Yaskawa INFORM job: u_tourne3TRJ1.JBI

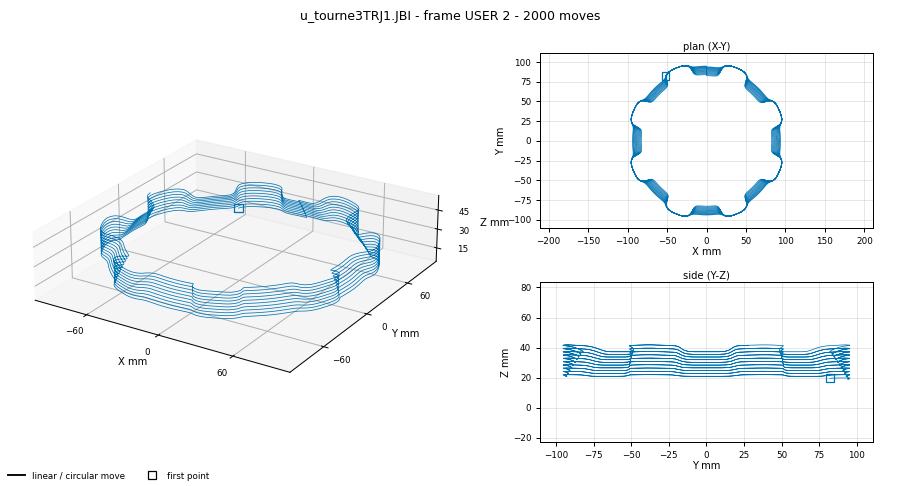
[picture p0: tool path of u_tourne3TRJ1.JBI in frame USER 2, 2000 of 2000 moves have a stored position in this frame; points joined in program order, loops and branches not executed]
/JOB
//NAME u_tourne3TRJ1
///FOLDERNAME DEMO
//POS
///NPOS 2000,0,2000,0,0,0
///USER 2
///TOOL 7
///POSTYPE USER
///RECTAN
///RCONF 1,0,0,0,0,0,0,0,0,0,0,0,0,0,0,0,0,0,0,0,0,0,0,0
C00000=-51.961,81.931,19.493,173.8545,9.2440,-3657.6170
C00001=-51.163,83.502,19.627,176.6033,6.2165,-3658.5035
C00002=-49.917,85.194,19.692,178.7206,4.0258,-3659.6330
C00003=-47.874,87.106,19.726,179.6780,1.7463,-3661.2065
C00004=-45.272,88.975,19.753,179.9712,0.2718,-3663.0322
C00005=-42.449,90.515,19.780,179.9981,0.0768,-3664.8747
C00006=-39.659,91.796,19.798,179.9970,0.0075,-3666.6340
C00007=-36.867,92.953,19.798,179.9968,0.0074,-3668.3657
C00008=-33.988,94.020,19.780,-179.9962,0.0778,-3670.1252
C00009=-30.903,94.927,19.753,-179.9766,0.2756,-3671.9676
C00010=-27.741,95.446,19.726,-179.6779,1.7445,-3673.7937
C00011=-24.945,95.538,19.692,-178.7208,4.0294,-3675.3667
C00012=-22.867,95.222,19.627,-176.6046,6.2189,-3676.4965
C00013=-21.192,94.676,19.493,-173.8561,9.2462,-3677.3831
C00014=-19.540,94.146,19.309,-171.9611,14.9094,-3678.2747
C00015=-17.528,93.824,19.120,-173.2655,21.6484,-3679.4181
C00016=-14.592,93.857,18.976,-177.3137,25.8724,-3681.1629
C00017=-10.190,94.262,18.917,-179.5911,27.0185,-3683.8301
C00018=-5.317,94.652,18.914,179.9702,27.0874,-3686.7848
C00019=0.000,94.804,18.916,-180.0000,27.0775,-3690.0000
C00020=0.000,93.772,20.859,-180.0000,28.8281,-3690.0000
C00021=5.223,93.624,20.857,-179.9587,28.8401,-3693.1930
C00022=10.031,93.243,20.860,179.4696,28.7637,-3696.1402
C00023=14.399,92.874,20.935,176.5083,27.4530,-3698.8129
C00024=17.292,92.935,21.118,171.4736,22.1760,-3700.5402
C00025=19.271,93.399,21.361,170.6019,14.0567,-3701.6582
C00026=20.902,94.108,21.598,173.3176,8.0331,-3702.5225
C00027=22.556,94.852,21.773,176.3408,5.3244,-3703.3766
C00028=24.607,95.353,21.858,178.5800,3.6143,-3704.4702
C00029=27.423,95.407,21.902,179.6582,1.5415,-3706.0363
C00030=30.651,94.973,21.938,179.9852,0.1578,-3707.8866
C00031=33.828,94.073,21.973,-179.9998,0.0671,-3709.7782
C00032=36.813,92.974,21.997,179.9979,0.0053,-3711.6011
C00033=39.712,91.773,21.997,-179.9970,0.0075,-3713.3991
C00034=42.599,90.440,21.973,179.9991,0.0692,-3715.2213
C00035=45.483,88.829,21.938,-179.9836,0.1565,-3717.1138
C00036=48.072,86.854,21.902,-179.6591,1.5379,-3718.9637
C00037=50.025,84.825,21.858,-178.5802,3.6128,-3720.5297
C00038=51.121,83.020,21.773,-176.3413,5.3283,-3721.6234
C00039=51.765,81.324,21.598,-173.3148,8.0333,-3722.4779
C00040=52.416,79.670,21.361,-170.5989,14.0579,-3723.3415
C00041=53.488,77.942,21.118,-171.4764,22.1779,-3724.4600
C00042=55.491,75.854,20.935,-176.5044,27.4539,-3726.1873
C00043=58.840,73.026,20.860,-179.4708,28.7627,-3728.8598
C00044=62.509,69.895,20.857,179.9582,28.8407,-3731.8071
C00045=66.307,66.307,20.859,180.0000,28.8305,-3735.0000
C00046=69.895,62.509,20.857,-179.9582,28.8407,-3738.1929
C00047=73.026,58.840,20.860,179.4708,28.7627,-3741.1402
C00048=75.854,55.491,20.935,176.5044,27.4539,-3743.8127
C00049=77.942,53.488,21.118,171.4764,22.1779,-3745.5400
C00050=79.670,52.416,21.361,170.5989,14.0579,-3746.6585
C00051=81.324,51.765,21.598,173.3148,8.0333,-3747.5221
C00052=83.020,51.121,21.773,176.3413,5.3283,-3748.3766
C00053=84.825,50.025,21.858,178.5802,3.6128,-3749.4703
C00054=86.854,48.072,21.902,179.6591,1.5379,-3751.0363
C00055=88.829,45.483,21.938,179.9836,0.1565,-3752.8862
C00056=90.440,42.599,21.973,-179.9991,0.0692,-3754.7787
C00057=91.773,39.712,21.997,179.9970,0.0075,-3756.6009
C00058=92.974,36.813,21.997,-179.9979,0.0053,-3758.3989
C00059=94.073,33.828,21.973,179.9998,0.0671,-3760.2218
C00060=94.973,30.651,21.938,-179.9852,0.1578,-3762.1134
C00061=95.407,27.423,21.902,-179.6582,1.5415,-3763.9637
C00062=95.353,24.607,21.858,-178.5800,3.6143,-3765.5298
C00063=94.852,22.556,21.773,-176.3408,5.3244,-3766.6234
C00064=94.108,20.902,21.598,-173.3176,8.0331,-3767.4775
C00065=93.399,19.271,21.361,-170.6019,14.0567,-3768.3418
C00066=92.935,17.292,21.118,-171.4736,22.1760,-3769.4598
C00067=92.874,14.399,20.935,-176.5083,27.4530,-3771.1871
C00068=93.243,10.031,20.860,-179.4696,28.7637,-3773.8598
C00069=93.624,5.223,20.857,179.9587,28.8401,-3776.8070
C00070=93.772,0.000,20.859,180.0000,28.8281,-3780.0000
C00071=93.624,-5.223,20.857,-179.9587,28.8401,-3783.1930
C00072=93.243,-10.031,20.860,179.4696,28.7637,-3786.1402
C00073=92.875,-14.399,20.935,176.5083,27.4530,-3788.8128
C00074=92.935,-17.292,21.118,171.4736,22.1760,-3790.5402
C00075=93.399,-19.271,21.361,170.6019,14.0567,-3791.6582
C00076=94.108,-20.902,21.598,173.3176,8.0331,-3792.5225
C00077=94.852,-22.556,21.773,176.3408,5.3244,-3793.3766
C00078=95.353,-24.607,21.858,178.5800,3.6143,-3794.4702
C00079=95.407,-27.423,21.902,179.6582,1.5415,-3796.0363
C00080=94.973,-30.651,21.938,179.9852,0.1578,-3797.8866
C00081=94.073,-33.828,21.973,-179.9998,0.0671,-3799.7782
C00082=92.974,-36.813,21.997,179.9979,0.0053,-3801.6011
C00083=91.773,-39.712,21.997,-179.9970,0.0075,-3803.3991
C00084=90.440,-42.599,21.973,179.9991,0.0692,-3805.2213
C00085=88.829,-45.483,21.938,-179.9836,0.1565,-3807.1138
C00086=86.854,-48.072,21.902,-179.6591,1.5379,-3808.9637
C00087=84.825,-50.025,21.858,-178.5802,3.6128,-3810.5297
C00088=83.020,-51.121,21.773,-176.3413,5.3283,-3811.6234
C00089=81.324,-51.765,21.598,-173.3148,8.0333,-3812.4779
C00090=79.670,-52.416,21.361,-170.5989,14.0579,-3813.3415
C00091=77.942,-53.488,21.118,-171.4764,22.1779,-3814.4600
C00092=75.854,-55.491,20.935,-176.5044,27.4539,-3816.1873
C00093=73.026,-58.840,20.860,-179.4708,28.7627,-3818.8598
C00094=69.895,-62.509,20.857,179.9582,28.8407,-3821.8071
C00095=66.307,-66.307,20.859,-180.0000,28.8305,-3825.0000
C00096=62.509,-69.895,20.857,-179.9582,28.8407,-3828.1929
C00097=58.840,-73.026,20.860,179.4708,28.7627,-3831.1402
C00098=55.491,-75.854,20.935,176.5044,27.4539,-3833.8127
C00099=53.488,-77.942,21.118,171.4764,22.1779,-3835.5400
C00100=52.416,-79.670,21.361,170.5989,14.0579,-3836.6585
C00101=51.765,-81.324,21.598,173.3148,8.0333,-3837.5221
C00102=51.121,-83.020,21.773,176.3413,5.3283,-3838.3766
C00103=50.025,-84.825,21.858,178.5802,3.6128,-3839.4703
C00104=48.072,-86.854,21.902,179.6591,1.5379,-3841.0363
C00105=45.483,-88.829,21.938,179.9836,0.1565,-3842.8862
C00106=42.599,-90.440,21.973,-179.9991,0.0692,-3844.7787
C00107=39.712,-91.773,21.997,179.9970,0.0075,-3846.6009
C00108=36.813,-92.974,21.997,-179.9979,0.0053,-3848.3989
C00109=33.828,-94.073,21.973,179.9998,0.0671,-3850.2218
C00110=30.651,-94.973,21.938,-179.9852,0.1578,-3852.1134
C00111=27.423,-95.407,21.902,-179.6582,1.5415,-3853.9637
C00112=24.607,-95.353,21.858,-178.5800,3.6143,-3855.5298
C00113=22.556,-94.852,21.773,-176.3408,5.3244,-3856.6234
C00114=20.902,-94.108,21.598,-173.3176,8.0331,-3857.4775
C00115=19.271,-93.399,21.361,-170.6019,14.0567,-3858.3418
C00116=17.292,-92.935,21.118,-171.4736,22.1760,-3859.4598
C00117=14.399,-92.874,20.935,-176.5083,27.4530,-3861.1871
C00118=10.031,-93.243,20.860,-179.4696,28.7637,-3863.8598
C00119=5.223,-93.624,20.857,179.9587,28.8401,-3866.8070
C00120=0.000,-93.772,20.859,-180.0000,28.8281,-3870.0000
C00121=0.000,-93.772,20.859,-180.0000,28.8281,-3870.0000
C00122=-5.223,-93.624,20.857,-179.9587,28.8401,-3873.1930
C00123=-10.031,-93.243,20.860,179.4696,28.7637,-3876.1402
C00124=-14.399,-92.875,20.935,176.5083,27.4530,-3878.8128
C00125=-17.292,-92.935,21.118,171.4736,22.1760,-3880.5402
C00126=-19.271,-93.399,21.361,170.6019,14.0567,-3881.6582
C00127=-20.902,-94.108,21.598,173.3176,8.0331,-3882.5225
C00128=-22.556,-94.852,21.773,176.3408,5.3244,-3883.3766
C00129=-24.607,-95.353,21.858,178.5800,3.6143,-3884.4702
C00130=-27.423,-95.407,21.902,179.6582,1.5415,-3886.0363
C00131=-30.651,-94.973,21.938,179.9852,0.1578,-3887.8866
C00132=-33.828,-94.073,21.973,-179.9998,0.0671,-3889.7782
C00133=-36.813,-92.974,21.997,179.9979,0.0053,-3891.6011
C00134=-39.712,-91.773,21.997,-179.9970,0.0075,-3893.3991
C00135=-42.599,-90.440,21.973,179.9991,0.0692,-3895.2213
C00136=-45.483,-88.829,21.938,-179.9836,0.1565,-3897.1138
C00137=-48.072,-86.854,21.902,-179.6591,1.5379,-3898.9637
C00138=-50.025,-84.825,21.858,-178.5802,3.6128,-3900.5297
C00139=-51.121,-83.020,21.773,-176.3413,5.3283,-3901.6234
C00140=-51.765,-81.324,21.598,-173.3148,8.0333,-3902.4779
C00141=-52.416,-79.670,21.361,-170.5989,14.0579,-3903.3415
C00142=-53.488,-77.942,21.118,-171.4764,22.1779,-3904.4600
C00143=-55.491,-75.854,20.935,-176.5044,27.4539,-3906.1873
C00144=-58.840,-73.026,20.860,-179.4708,28.7627,-3908.8598
C00145=-62.509,-69.895,20.857,179.9582,28.8407,-3911.8071
C00146=-66.307,-66.307,20.859,-180.0000,28.8305,-3915.0000
C00147=-69.895,-62.509,20.857,-179.9582,28.8407,-3918.1929
C00148=-73.026,-58.840,20.860,179.4708,28.7627,-3921.1402
C00149=-75.854,-55.491,20.935,176.5044,27.4539,-3923.8127
C00150=-77.942,-53.488,21.118,171.4764,22.1779,-3925.5400
C00151=-79.670,-52.416,21.361,170.5989,14.0579,-3926.6585
C00152=-81.324,-51.765,21.598,173.3148,8.0333,-3927.5221
C00153=-83.020,-51.121,21.773,176.3413,5.3283,-3928.3766
C00154=-84.825,-50.025,21.858,178.5802,3.6128,-3929.4703
C00155=-86.854,-48.072,21.902,179.6591,1.5379,-3931.0363
C00156=-88.829,-45.483,21.938,179.9836,0.1565,-3932.8862
C00157=-90.440,-42.599,21.973,-179.9991,0.0692,-3934.7787
C00158=-91.773,-39.712,21.997,179.9970,0.0075,-3936.6009
C00159=-92.974,-36.813,21.997,-179.9979,0.0053,-3938.3989
C00160=-94.073,-33.828,21.973,179.9998,0.0671,-3940.2218
C00161=-94.973,-30.651,21.938,-179.9852,0.1578,-3942.1134
C00162=-95.407,-27.423,21.902,-179.6582,1.5415,-3943.9637
C00163=-95.353,-24.607,21.858,-178.5800,3.6143,-3945.5298
C00164=-94.852,-22.556,21.773,-176.3408,5.3244,-3946.6234
C00165=-94.108,-20.902,21.598,-173.3176,8.0331,-3947.4775
C00166=-93.399,-19.271,21.361,-170.6019,14.0567,-3948.3418
C00167=-92.935,-17.292,21.118,-171.4736,22.1760,-3949.4598
C00168=-92.874,-14.399,20.935,-176.5083,27.4530,-3951.1871
C00169=-93.243,-10.031,20.860,-179.4696,28.7637,-3953.8598
C00170=-93.624,-5.223,20.857,179.9587,28.8401,-3956.8070
C00171=-93.772,0.000,20.859,180.0000,28.8281,-3960.0000
C00172=-93.624,5.223,20.857,-179.9587,28.8401,-3963.1930
C00173=-93.243,10.031,20.860,179.4696,28.7637,-3966.1402
C00174=-92.875,14.399,20.935,176.5083,27.4530,-3968.8128
C00175=-92.935,17.292,21.118,171.4736,22.1760,-3970.5402
C00176=-93.399,19.271,21.361,170.6019,14.0567,-3971.6582
C00177=-94.108,20.902,21.598,173.3176,8.0331,-3972.5225
C00178=-94.852,22.556,21.773,176.3408,5.3244,-3973.3766
C00179=-95.353,24.607,21.858,178.5800,3.6143,-3974.4702
C00180=-95.407,27.423,21.902,179.6582,1.5415,-3976.0363
C00181=-94.973,30.651,21.938,179.9852,0.1578,-3977.8866
C00182=-94.073,33.828,21.973,-179.9998,0.0671,-3979.7782
C00183=-92.974,36.813,21.997,179.9979,0.0053,-3981.6011
C00184=-91.773,39.712,21.997,-179.9970,0.0075,-3983.3991
C00185=-90.440,42.599,21.973,179.9991,0.0692,-3985.2213
C00186=-88.829,45.483,21.938,-179.9836,0.1565,-3987.1138
C00187=-86.854,48.072,21.902,-179.6591,1.5379,-3988.9637
C00188=-84.825,50.025,21.858,-178.5802,3.6128,-3990.5297
C00189=-83.020,51.121,21.773,-176.3413,5.3283,-3991.6234
C00190=-81.324,51.765,21.598,-173.3148,8.0333,-3992.4779
C00191=-79.670,52.416,21.361,-170.5989,14.0579,-3993.3415
C00192=-77.942,53.488,21.118,-171.4764,22.1779,-3994.4600
C00193=-75.854,55.491,20.935,-176.5044,27.4539,-3996.1873
C00194=-73.026,58.840,20.860,-179.4708,28.7627,-3998.8598
C00195=-69.895,62.509,20.857,179.9582,28.8407,-4001.8071
C00196=-66.307,66.307,20.859,180.0000,28.8305,-4005.0000
C00197=-62.509,69.895,20.857,-179.9582,28.8407,-4008.1929
C00198=-58.840,73.026,20.860,179.4708,28.7627,-4011.1402
C00199=-55.491,75.854,20.935,176.5044,27.4539,-4013.8127
C00200=-53.488,77.942,21.118,171.4764,22.1779,-4015.5400
C00201=-52.416,79.670,21.361,170.5989,14.0579,-4016.6585
C00202=-51.765,81.324,21.598,173.3148,8.0333,-4017.5221
C00203=-51.121,83.020,21.773,176.3413,5.3283,-4018.3766
C00204=-50.025,84.825,21.858,178.5802,3.6128,-4019.4703
C00205=-48.072,86.854,21.902,179.6591,1.5379,-4021.0363
C00206=-45.483,88.829,21.938,179.9836,0.1565,-4022.8862
C00207=-42.599,90.440,21.973,-179.9991,0.0692,-4024.7787
C00208=-39.712,91.773,21.997,179.9970,0.0075,-4026.6009
C00209=-36.813,92.974,21.997,-179.9979,0.0053,-4028.3989
C00210=-33.828,94.073,21.973,179.9998,0.0671,-4030.2218
C00211=-30.651,94.973,21.938,-179.9852,0.1578,-4032.1134
C00212=-27.423,95.407,21.902,-179.6582,1.5415,-4033.9637
C00213=-24.607,95.353,21.858,-178.5800,3.6143,-4035.5298
C00214=-22.556,94.852,21.773,-176.3408,5.3244,-4036.6234
C00215=-20.902,94.108,21.598,-173.3176,8.0331,-4037.4775
C00216=-19.271,93.399,21.361,-170.6019,14.0567,-4038.3418
C00217=-17.292,92.935,21.118,-171.4736,22.1760,-4039.4598
C00218=-14.399,92.875,20.935,-176.5083,27.4530,-4041.1872
C00219=-10.031,93.243,20.860,-179.4696,28.7637,-4043.8598
C00220=-5.223,93.624,20.857,179.9587,28.8401,-4046.8070
C00221=0.000,93.772,20.859,-180.0000,28.8281,-4050.0000
C00222=0.000,92.684,22.771,-180.0000,30.3909,-4050.0000
C00223=5.124,92.540,22.769,-179.9518,30.3994,-4053.1693
C00224=9.864,92.169,22.773,179.3255,30.3134,-4056.1086
C00225=14.194,91.838,22.865,175.6033,28.8062,-4058.7858
C00226=17.042,91.994,23.091,169.6619,22.2216,-4060.4951
C00227=18.986,92.606,23.393,169.6266,12.7358,-4061.5862
C00228=20.592,93.503,23.691,173.2393,6.5920,-4062.4199
C00229=22.223,94.456,23.912,176.4053,4.2313,-4063.2394
C00230=24.245,95.156,24.019,178.5515,3.0336,-4064.2944
C00231=27.082,95.366,24.075,179.6706,1.2647,-4065.8535
C00232=30.380,95.022,24.120,179.9985,0.0236,-4067.7299
C00233=33.658,94.129,24.166,179.9969,0.0597,-4069.6757
C00234=36.755,92.996,24.196,179.9979,0.0053,-4071.5655
C00235=39.769,91.748,24.196,179.9977,0.0053,-4073.4348
C00236=42.760,90.359,24.166,179.9987,0.0564,-4075.3246
C00237=45.709,88.673,24.120,-179.9977,0.0205,-4077.2701
C00238=48.284,86.584,24.075,-179.6697,1.2668,-4079.1464
C00239=50.142,84.429,24.019,-178.5525,3.0331,-4080.7059
C00240=51.076,82.504,23.912,-176.4065,4.2307,-4081.7605
C00241=51.556,80.678,23.691,-173.2418,6.5908,-4082.5800
C00242=52.057,78.907,23.393,-169.6292,12.7370,-4083.4139
C00243=52.999,77.101,23.091,-169.6605,22.2236,-4084.5045
C00244=54.903,74.976,22.865,-175.5993,28.8036,-4086.2144
C00245=58.198,72.148,22.773,-179.3268,30.3167,-4088.8913
C00246=61.813,69.059,22.769,179.9465,30.4010,-4091.8309
C00247=65.538,65.538,22.771,-180.0000,30.3891,-4095.0000
C00248=69.059,61.813,22.769,-179.9465,30.4010,-4098.1691
C00249=72.148,58.198,22.773,179.3268,30.3167,-4101.1087
C00250=74.976,54.903,22.865,175.6032,28.8076,-4103.7856
C00251=77.101,52.999,23.091,169.6605,22.2236,-4105.4955
C00252=78.907,52.057,23.393,169.6292,12.7370,-4106.5861
C00253=80.678,51.556,23.691,173.2418,6.5908,-4107.4200
C00254=82.504,51.076,23.912,176.4065,4.2307,-4108.2395
C00255=84.429,50.142,24.019,178.5525,3.0331,-4109.2941
C00256=86.584,48.284,24.075,179.6697,1.2668,-4110.8536
C00257=88.673,45.709,24.120,179.9977,0.0205,-4112.7299
C00258=90.359,42.760,24.166,-179.9987,0.0564,-4114.6754
C00259=91.748,39.769,24.196,-179.9977,0.0053,-4116.5652
C00260=92.996,36.755,24.196,-179.9979,0.0053,-4118.4345
C00261=94.129,33.658,24.166,-179.9969,0.0597,-4120.3243
C00262=95.022,30.380,24.120,-179.9985,0.0236,-4122.2701
C00263=95.366,27.082,24.075,-179.6706,1.2647,-4124.1465
C00264=95.156,24.245,24.019,-178.5515,3.0336,-4125.7056
C00265=94.456,22.223,23.912,-176.4053,4.2313,-4126.7606
C00266=93.503,20.592,23.691,-173.2393,6.5920,-4127.5801
C00267=92.606,18.986,23.393,-169.6266,12.7358,-4128.4138
C00268=91.994,17.042,23.091,-169.6619,22.2216,-4129.5049
C00269=91.838,14.194,22.865,-175.6033,28.8062,-4131.2142
C00270=92.169,9.864,22.773,-179.3255,30.3134,-4133.8914
C00271=92.540,5.124,22.769,179.9518,30.3994,-4136.8307
C00272=92.684,0.000,22.771,-180.0000,30.3909,-4140.0000
C00273=92.540,-5.124,22.769,-179.9518,30.3994,-4143.1693
C00274=92.169,-9.864,22.773,179.3255,30.3134,-4146.1086
C00275=91.838,-14.194,22.865,175.6033,28.8062,-4148.7858
C00276=91.994,-17.042,23.091,169.6619,22.2216,-4150.4951
C00277=92.606,-18.986,23.393,169.6266,12.7358,-4151.5862
C00278=93.503,-20.592,23.691,173.2393,6.5920,-4152.4199
C00279=94.456,-22.223,23.912,176.4053,4.2313,-4153.2394
C00280=95.156,-24.245,24.019,178.5515,3.0336,-4154.2944
C00281=95.366,-27.082,24.075,179.6706,1.2647,-4155.8535
C00282=95.022,-30.380,24.120,179.9985,0.0236,-4157.7299
C00283=94.129,-33.658,24.166,179.9969,0.0597,-4159.6757
C00284=92.996,-36.755,24.196,179.9979,0.0053,-4161.5655
C00285=91.748,-39.769,24.196,179.9977,0.0053,-4163.4348
C00286=90.359,-42.760,24.166,179.9987,0.0564,-4165.3246
C00287=88.673,-45.709,24.120,-179.9977,0.0205,-4167.2701
C00288=86.584,-48.284,24.075,-179.6697,1.2668,-4169.1464
C00289=84.429,-50.142,24.019,-178.5525,3.0331,-4170.7059
C00290=82.504,-51.076,23.912,-176.4065,4.2307,-4171.7605
C00291=80.678,-51.556,23.691,-173.2418,6.5908,-4172.5800
C00292=78.907,-52.057,23.393,-169.6292,12.7370,-4173.4139
C00293=77.101,-52.999,23.091,-169.6605,22.2236,-4174.5045
C00294=74.976,-54.903,22.865,-175.5993,28.8036,-4176.2144
C00295=72.148,-58.198,22.773,-179.3268,30.3167,-4178.8913
C00296=69.059,-61.813,22.769,179.9465,30.4010,-4181.8309
C00297=65.538,-65.538,22.771,180.0000,30.3891,-4185.0000
C00298=61.813,-69.059,22.769,-179.9465,30.4010,-4188.1691
C00299=58.198,-72.148,22.773,179.3268,30.3167,-4191.1087
C00300=54.903,-74.976,22.865,175.6032,28.8076,-4193.7856
C00301=52.999,-77.101,23.091,169.6605,22.2236,-4195.4955
C00302=52.057,-78.907,23.393,169.6292,12.7370,-4196.5861
C00303=51.556,-80.678,23.691,173.2418,6.5908,-4197.4200
C00304=51.076,-82.504,23.912,176.4065,4.2307,-4198.2395
C00305=50.142,-84.429,24.019,178.5525,3.0331,-4199.2941
C00306=48.284,-86.584,24.075,179.6697,1.2668,-4200.8536
C00307=45.709,-88.673,24.120,179.9977,0.0205,-4202.7299
C00308=42.760,-90.359,24.166,-179.9987,0.0564,-4204.6754
C00309=39.769,-91.748,24.196,-179.9977,0.0053,-4206.5652
C00310=36.755,-92.996,24.196,-179.9979,0.0053,-4208.4345
C00311=33.658,-94.129,24.166,-179.9969,0.0597,-4210.3243
C00312=30.380,-95.022,24.120,-179.9985,0.0236,-4212.2701
C00313=27.082,-95.366,24.075,-179.6706,1.2647,-4214.1465
C00314=24.245,-95.156,24.019,-178.5515,3.0336,-4215.7056
C00315=22.223,-94.456,23.912,-176.4053,4.2313,-4216.7606
C00316=20.592,-93.503,23.691,-173.2393,6.5920,-4217.5801
C00317=18.986,-92.606,23.393,-169.6266,12.7358,-4218.4138
C00318=17.042,-91.994,23.091,-169.6619,22.2216,-4219.5049
C00319=14.194,-91.838,22.865,-175.6033,28.8062,-4221.2142
C00320=9.864,-92.169,22.773,-179.3255,30.3134,-4223.8914
C00321=5.124,-92.540,22.769,179.9518,30.3994,-4226.8307
C00322=0.000,-92.684,22.771,180.0000,30.3909,-4230.0000
C00323=0.000,-92.684,22.771,180.0000,30.3909,-4230.0000
C00324=-5.124,-92.540,22.769,-179.9518,30.3994,-4233.1693
C00325=-9.864,-92.169,22.773,179.3255,30.3134,-4236.1086
C00326=-14.194,-91.838,22.865,175.6033,28.8062,-4238.7858
C00327=-17.042,-91.994,23.091,169.6619,22.2216,-4240.4951
C00328=-18.986,-92.606,23.393,169.6266,12.7358,-4241.5862
C00329=-20.592,-93.503,23.691,173.2393,6.5920,-4242.4199
C00330=-22.223,-94.456,23.912,176.4053,4.2313,-4243.2394
C00331=-24.245,-95.156,24.019,178.5515,3.0336,-4244.2944
C00332=-27.082,-95.366,24.075,179.6706,1.2647,-4245.8535
C00333=-30.380,-95.022,24.120,179.9985,0.0236,-4247.7299
C00334=-33.658,-94.129,24.166,179.9969,0.0597,-4249.6757
C00335=-36.755,-92.996,24.196,179.9979,0.0053,-4251.5655
C00336=-39.769,-91.748,24.196,179.9977,0.0053,-4253.4348
C00337=-42.760,-90.359,24.166,179.9987,0.0564,-4255.3246
C00338=-45.709,-88.673,24.120,-179.9977,0.0205,-4257.2701
C00339=-48.284,-86.584,24.075,-179.6697,1.2668,-4259.1464
C00340=-50.142,-84.429,24.019,-178.5525,3.0331,-4260.7059
C00341=-51.076,-82.504,23.912,-176.4065,4.2307,-4261.7605
C00342=-51.556,-80.678,23.691,-173.2418,6.5908,-4262.5800
C00343=-52.057,-78.907,23.393,-169.6292,12.7370,-4263.4139
C00344=-52.999,-77.101,23.091,-169.6605,22.2236,-4264.5045
C00345=-54.903,-74.976,22.865,-175.5993,28.8036,-4266.2144
C00346=-58.198,-72.148,22.773,-179.3268,30.3167,-4268.8913
C00347=-61.813,-69.059,22.769,179.9465,30.4010,-4271.8309
C00348=-65.538,-65.538,22.771,-180.0000,30.3891,-4275.0000
C00349=-69.059,-61.813,22.769,-179.9465,30.4010,-4278.1691
C00350=-72.148,-58.198,22.773,179.3268,30.3167,-4281.1087
C00351=-74.976,-54.903,22.865,175.6032,28.8076,-4283.7856
C00352=-77.101,-52.999,23.091,169.6605,22.2236,-4285.4955
C00353=-78.907,-52.057,23.393,169.6292,12.7370,-4286.5861
C00354=-80.678,-51.556,23.691,173.2418,6.5908,-4287.4200
C00355=-82.504,-51.076,23.912,176.4065,4.2307,-4288.2395
C00356=-84.429,-50.142,24.019,178.5525,3.0331,-4289.2941
C00357=-86.584,-48.284,24.075,179.6697,1.2668,-4290.8536
C00358=-88.673,-45.709,24.120,179.9977,0.0205,-4292.7299
C00359=-90.359,-42.760,24.166,-179.9987,0.0564,-4294.6754
C00360=-91.748,-39.769,24.196,-179.9977,0.0053,-4296.5652
C00361=-92.996,-36.755,24.196,-179.9979,0.0053,-4298.4345
C00362=-94.129,-33.658,24.166,-179.9969,0.0597,-4300.3243
C00363=-95.022,-30.380,24.120,-179.9985,0.0236,-4302.2701
C00364=-95.366,-27.082,24.075,-179.6706,1.2647,-4304.1465
C00365=-95.156,-24.245,24.019,-178.5515,3.0336,-4305.7056
C00366=-94.456,-22.223,23.912,-176.4053,4.2313,-4306.7606
C00367=-93.503,-20.592,23.691,-173.2393,6.5920,-4307.5801
C00368=-92.606,-18.986,23.393,-169.6266,12.7358,-4308.4138
C00369=-91.994,-17.042,23.091,-169.6619,22.2216,-4309.5049
C00370=-91.838,-14.194,22.865,-175.6033,28.8062,-4311.2142
C00371=-92.169,-9.864,22.773,-179.3255,30.3134,-4313.8914
C00372=-92.540,-5.124,22.769,179.9518,30.3994,-4316.8307
C00373=-92.684,0.000,22.771,-180.0000,30.3909,-4320.0000
C00374=-92.540,5.124,22.769,-179.9518,30.3994,-4323.1693
C00375=-92.169,9.864,22.773,179.3255,30.3134,-4326.1086
C00376=-91.838,14.194,22.865,175.6033,28.8062,-4328.7858
C00377=-91.994,17.042,23.091,169.6619,22.2216,-4330.4951
C00378=-92.606,18.986,23.393,169.6266,12.7358,-4331.5862
C00379=-93.503,20.592,23.691,173.2393,6.5920,-4332.4199
C00380=-94.456,22.223,23.912,176.4053,4.2313,-4333.2394
C00381=-95.156,24.245,24.019,178.5515,3.0336,-4334.2944
C00382=-95.366,27.082,24.075,179.6706,1.2647,-4335.8535
C00383=-95.022,30.380,24.120,179.9985,0.0236,-4337.7299
C00384=-94.129,33.658,24.166,179.9969,0.0597,-4339.6757
C00385=-92.996,36.755,24.196,179.9979,0.0053,-4341.5655
C00386=-91.748,39.769,24.196,179.9977,0.0053,-4343.4348
C00387=-90.359,42.760,24.166,179.9987,0.0564,-4345.3246
C00388=-88.673,45.709,24.120,-179.9977,0.0205,-4347.2701
C00389=-86.584,48.284,24.075,-179.6697,1.2668,-4349.1464
C00390=-84.429,50.142,24.019,-178.5525,3.0331,-4350.7059
C00391=-82.504,51.076,23.912,-176.4065,4.2307,-4351.7605
C00392=-80.678,51.556,23.691,-173.2418,6.5908,-4352.5800
C00393=-78.907,52.057,23.393,-169.6292,12.7370,-4353.4139
C00394=-77.101,52.999,23.091,-169.6605,22.2236,-4354.5045
C00395=-74.976,54.903,22.865,-175.5993,28.8036,-4356.2144
C00396=-72.148,58.198,22.773,-179.3268,30.3167,-4358.8913
C00397=-69.059,61.813,22.769,179.9465,30.4010,-4361.8309
C00398=-65.538,65.538,22.771,-180.0000,30.3891,-4365.0000
C00399=-61.813,69.059,22.769,-179.9465,30.4010,-4368.1691
C00400=-58.198,72.148,22.773,179.3268,30.3167,-4371.1087
C00401=-54.903,74.976,22.865,175.6032,28.8076,-4373.7856
C00402=-52.999,77.101,23.091,169.6605,22.2236,-4375.4955
C00403=-52.057,78.907,23.393,169.6292,12.7370,-4376.5861
C00404=-51.556,80.678,23.691,173.2418,6.5908,-4377.4200
C00405=-51.076,82.504,23.912,176.4065,4.2307,-4378.2395
C00406=-50.142,84.429,24.019,178.5525,3.0331,-4379.2941
C00407=-48.284,86.584,24.075,179.6697,1.2668,-4380.8536
C00408=-45.709,88.673,24.120,179.9977,0.0205,-4382.7299
C00409=-42.760,90.359,24.166,-179.9987,0.0564,-4384.6754
C00410=-39.769,91.748,24.196,-179.9977,0.0053,-4386.5652
C00411=-36.755,92.996,24.196,-179.9979,0.0053,-4388.4345
C00412=-33.658,94.129,24.166,-179.9969,0.0597,-4390.3243
C00413=-30.380,95.022,24.120,-179.9985,0.0236,-4392.2701
C00414=-27.082,95.366,24.075,-179.6706,1.2647,-4394.1465
C00415=-24.245,95.156,24.019,-178.5515,3.0336,-4395.7056
C00416=-22.223,94.456,23.912,-176.4053,4.2313,-4396.7606
C00417=-20.592,93.503,23.691,-173.2393,6.5920,-4397.5801
C00418=-18.986,92.606,23.393,-169.6266,12.7358,-4398.4138
C00419=-17.042,91.994,23.091,-169.6619,22.2216,-4399.5049
C00420=-14.194,91.838,22.865,-175.6033,28.8062,-4401.2142
C00421=-9.864,92.169,22.773,-179.3255,30.3134,-4403.8914
C00422=-5.124,92.540,22.769,179.9518,30.3994,-4406.8307
C00423=0.000,92.684,22.771,-180.0000,30.3909,-4410.0000
C00424=0.000,91.548,24.655,-180.0000,31.7764,-4410.0000
C00425=5.020,91.408,24.652,-179.9386,31.7913,-4413.1434
C00426=9.690,91.047,24.657,179.1672,31.6940,-4416.0750
C00427=13.981,90.755,24.767,174.6081,29.9498,-4418.7577
C00428=16.781,91.008,25.041,167.9432,21.7872,-4420.4474
C00429=18.686,91.772,25.406,169.1360,11.0995,-4421.5089
C00430=20.265,92.865,25.771,173.6100,5.1205,-4422.3101
C00431=21.871,94.037,26.043,176.8157,3.0731,-4423.0930
C00432=23.861,94.948,26.175,178.6786,2.3162,-4424.1066
C00433=26.720,95.323,26.245,179.7166,0.9262,-4425.6587
C00434=30.093,95.074,26.301,-179.9821,-0.1326,-4427.5637
C00435=33.476,94.189,26.358,-179.9972,0.0435,-4429.5659
C00436=36.693,93.020,26.395,179.9979,0.0053,-4431.5274
C00437=39.829,91.721,26.395,179.9977,0.0053,-4433.4725
C00438=42.931,90.273,26.358,179.9983,0.0436,-4435.4343
C00439=45.948,88.507,26.301,179.9790,-0.1336,-4437.4359
C00440=48.509,86.297,26.245,-179.7191,0.9269,-4439.3411
C00441=50.266,84.010,26.175,-178.6733,2.3167,-4440.8935
C00442=51.029,81.959,26.043,-176.8139,3.0727,-4441.9071
C00443=51.336,79.995,25.771,-173.6111,5.1213,-4442.6899
C00444=51.679,78.105,25.406,-169.1359,11.0962,-4443.4910
C00445=52.487,76.218,25.041,-167.9434,21.7869,-4444.5530
C00446=54.287,74.059,24.767,-174.6079,29.9481,-4446.2423
C00447=57.528,71.231,24.657,-179.1658,31.6931,-4448.9252
C00448=61.085,68.184,24.652,179.9356,31.7887,-4451.8567
C00449=64.734,64.734,24.655,180.0000,31.7790,-4455.0000
C00450=68.184,61.085,24.652,-179.9356,31.7887,-4458.1433
C00451=71.231,57.528,24.657,179.1658,31.6931,-4461.0748
C00452=74.059,54.287,24.767,174.6079,29.9481,-4463.7577
C00453=76.218,52.487,25.041,167.9434,21.7869,-4465.4470
C00454=78.105,51.679,25.406,169.1359,11.0962,-4466.5090
C00455=79.995,51.336,25.771,173.6111,5.1213,-4467.3101
C00456=81.959,51.029,26.043,176.8139,3.0727,-4468.0929
C00457=84.010,50.266,26.175,178.6733,2.3167,-4469.1065
C00458=86.297,48.509,26.245,179.7191,0.9269,-4470.6589
C00459=88.507,45.948,26.301,-179.9790,-0.1336,-4472.5641
C00460=90.273,42.931,26.358,-179.9983,0.0436,-4474.5657
C00461=91.721,39.829,26.395,-179.9977,0.0053,-4476.5275
C00462=93.020,36.693,26.395,-179.9979,0.0053,-4478.4726
C00463=94.189,33.476,26.358,179.9972,0.0435,-4480.4341
C00464=95.074,30.093,26.301,179.9821,-0.1326,-4482.4363
C00465=95.323,26.720,26.245,-179.7166,0.9262,-4484.3413
C00466=94.948,23.861,26.175,-178.6786,2.3162,-4485.8934
C00467=94.037,21.871,26.043,-176.8157,3.0731,-4486.9070
C00468=92.865,20.265,25.771,-173.6100,5.1205,-4487.6899
C00469=91.772,18.686,25.406,-169.1360,11.0995,-4488.4911
C00470=91.008,16.781,25.041,-167.9432,21.7872,-4489.5526
C00471=90.755,13.981,24.767,-174.6081,29.9498,-4491.2423
C00472=91.047,9.690,24.657,-179.1672,31.6940,-4493.9250
C00473=91.408,5.020,24.652,179.9386,31.7913,-4496.8566
C00474=91.548,0.000,24.655,180.0000,31.7764,-4500.0000
C00475=91.408,-5.020,24.652,-179.9386,31.7913,-4503.1434
C00476=91.047,-9.690,24.657,179.1672,31.6940,-4506.0750
C00477=90.755,-13.981,24.767,174.6081,29.9498,-4508.7577
C00478=91.008,-16.781,25.041,167.9432,21.7872,-4510.4474
C00479=91.772,-18.686,25.406,169.1360,11.0995,-4511.5089
C00480=92.865,-20.265,25.771,173.6100,5.1205,-4512.3101
C00481=94.037,-21.871,26.043,176.8157,3.0731,-4513.0930
C00482=94.948,-23.861,26.175,178.6786,2.3162,-4514.1066
C00483=95.323,-26.720,26.245,179.7166,0.9262,-4515.6587
C00484=95.074,-30.093,26.301,-179.9821,-0.1326,-4517.5637
C00485=94.189,-33.476,26.358,-179.9972,0.0435,-4519.5659
C00486=93.020,-36.693,26.395,179.9979,0.0053,-4521.5274
C00487=91.721,-39.829,26.395,179.9977,0.0053,-4523.4725
C00488=90.273,-42.931,26.358,179.9983,0.0436,-4525.4343
C00489=88.507,-45.948,26.301,179.9790,-0.1336,-4527.4359
C00490=86.297,-48.509,26.245,-179.7191,0.9269,-4529.3411
C00491=84.010,-50.266,26.175,-178.6733,2.3167,-4530.8935
C00492=81.959,-51.029,26.043,-176.8139,3.0727,-4531.9071
C00493=79.995,-51.336,25.771,-173.6111,5.1213,-4532.6899
C00494=78.105,-51.679,25.406,-169.1359,11.0962,-4533.4910
C00495=76.218,-52.487,25.041,-167.9434,21.7869,-4534.5530
C00496=74.059,-54.287,24.767,-174.6079,29.9481,-4536.2423
C00497=71.231,-57.528,24.657,-179.1658,31.6931,-4538.9252
C00498=68.184,-61.085,24.652,179.9356,31.7887,-4541.8567
C00499=64.734,-64.734,24.655,-180.0000,31.7790,-4545.0000
C00500=61.085,-68.184,24.652,-179.9356,31.7887,-4548.1433
C00501=57.528,-71.231,24.657,179.1658,31.6931,-4551.0748
C00502=54.287,-74.059,24.767,174.6079,29.9481,-4553.7577
C00503=52.487,-76.218,25.041,167.9434,21.7869,-4555.4470
C00504=51.679,-78.105,25.406,169.1359,11.0962,-4556.5090
C00505=51.336,-79.995,25.771,173.6111,5.1213,-4557.3101
C00506=51.029,-81.959,26.043,176.8139,3.0727,-4558.0929
C00507=50.266,-84.010,26.175,178.6733,2.3167,-4559.1065
C00508=48.509,-86.297,26.245,179.7191,0.9269,-4560.6589
C00509=45.948,-88.507,26.301,-179.9790,-0.1336,-4562.5641
C00510=42.931,-90.273,26.358,-179.9983,0.0436,-4564.5657
C00511=39.829,-91.721,26.395,-179.9977,0.0053,-4566.5275
C00512=36.693,-93.020,26.395,-179.9979,0.0053,-4568.4726
C00513=33.476,-94.189,26.358,179.9972,0.0435,-4570.4341
C00514=30.093,-95.074,26.301,179.9821,-0.1326,-4572.4363
C00515=26.720,-95.323,26.245,-179.7166,0.9262,-4574.3413
C00516=23.861,-94.948,26.175,-178.6786,2.3162,-4575.8934
C00517=21.871,-94.037,26.043,-176.8157,3.0731,-4576.9070
C00518=20.265,-92.865,25.771,-173.6100,5.1205,-4577.6899
C00519=18.686,-91.772,25.406,-169.1360,11.0995,-4578.4911
C00520=16.781,-91.008,25.041,-167.9432,21.7872,-4579.5526
C00521=13.981,-90.755,24.767,-174.6081,29.9498,-4581.2423
C00522=9.690,-91.047,24.657,-179.1672,31.6940,-4583.9250
C00523=5.020,-91.408,24.652,179.9386,31.7913,-4586.8566
C00524=0.000,-91.548,24.655,-180.0000,31.7764,-4590.0000
C00525=0.000,-91.548,24.655,-180.0000,31.7764,-4590.0000
C00526=-5.020,-91.408,24.652,-179.9386,31.7913,-4593.1434
C00527=-9.690,-91.047,24.657,179.1672,31.6940,-4596.0750
C00528=-13.981,-90.755,24.767,174.6081,29.9498,-4598.7577
C00529=-16.781,-91.008,25.041,167.9432,21.7872,-4600.4474
C00530=-18.686,-91.772,25.406,169.1360,11.0995,-4601.5089
C00531=-20.265,-92.865,25.771,173.6100,5.1205,-4602.3101
C00532=-21.871,-94.037,26.043,176.8157,3.0731,-4603.0930
C00533=-23.861,-94.948,26.175,178.6786,2.3162,-4604.1066
C00534=-26.720,-95.323,26.245,179.7166,0.9262,-4605.6587
C00535=-30.093,-95.074,26.301,-179.9821,-0.1326,-4607.5637
C00536=-33.476,-94.189,26.358,-179.9972,0.0435,-4609.5659
C00537=-36.693,-93.020,26.395,179.9979,0.0053,-4611.5274
C00538=-39.829,-91.721,26.395,179.9977,0.0053,-4613.4725
C00539=-42.931,-90.273,26.358,179.9983,0.0436,-4615.4343
C00540=-45.948,-88.507,26.301,179.9790,-0.1336,-4617.4359
C00541=-48.509,-86.297,26.245,-179.7191,0.9269,-4619.3411
C00542=-50.266,-84.010,26.175,-178.6733,2.3167,-4620.8935
C00543=-51.029,-81.959,26.043,-176.8139,3.0727,-4621.9071
C00544=-51.336,-79.995,25.771,-173.6111,5.1213,-4622.6899
C00545=-51.679,-78.105,25.406,-169.1359,11.0962,-4623.4910
C00546=-52.487,-76.218,25.041,-167.9434,21.7869,-4624.5530
C00547=-54.287,-74.059,24.767,-174.6079,29.9481,-4626.2423
C00548=-57.528,-71.231,24.657,-179.1658,31.6931,-4628.9252
C00549=-61.085,-68.184,24.652,179.9356,31.7887,-4631.8567
C00550=-64.734,-64.734,24.655,-180.0000,31.7790,-4635.0000
C00551=-68.184,-61.085,24.652,-179.9356,31.7887,-4638.1433
C00552=-71.231,-57.528,24.657,179.1658,31.6931,-4641.0748
C00553=-74.059,-54.287,24.767,174.6079,29.9481,-4643.7577
C00554=-76.218,-52.487,25.041,167.9434,21.7869,-4645.4470
C00555=-78.105,-51.679,25.406,169.1359,11.0962,-4646.5090
C00556=-79.995,-51.336,25.771,173.6111,5.1213,-4647.3101
C00557=-81.959,-51.029,26.043,176.8139,3.0727,-4648.0929
C00558=-84.010,-50.266,26.175,178.6733,2.3167,-4649.1065
C00559=-86.297,-48.509,26.245,179.7191,0.9269,-4650.6589
C00560=-88.507,-45.948,26.301,-179.9790,-0.1336,-4652.5641
C00561=-90.273,-42.931,26.358,-179.9983,0.0436,-4654.5657
C00562=-91.721,-39.829,26.395,-179.9977,0.0053,-4656.5275
C00563=-93.020,-36.693,26.395,-179.9979,0.0053,-4658.4726
C00564=-94.189,-33.476,26.358,179.9972,0.0435,-4660.4341
C00565=-95.074,-30.093,26.301,179.9821,-0.1326,-4662.4363
C00566=-95.323,-26.720,26.245,-179.7166,0.9262,-4664.3413
C00567=-94.948,-23.861,26.175,-178.6786,2.3162,-4665.8934
C00568=-94.037,-21.871,26.043,-176.8157,3.0731,-4666.9070
C00569=-92.865,-20.265,25.771,-173.6100,5.1205,-4667.6899
C00570=-91.772,-18.686,25.406,-169.1360,11.0995,-4668.4911
C00571=-91.008,-16.781,25.041,-167.9432,21.7872,-4669.5526
C00572=-90.755,-13.981,24.767,-174.6081,29.9498,-4671.2423
C00573=-91.047,-9.690,24.657,-179.1672,31.6940,-4673.9250
C00574=-91.408,-5.020,24.652,179.9386,31.7913,-4676.8566
C00575=-91.548,0.000,24.655,180.0000,31.7764,-4680.0000
C00576=-91.408,5.020,24.652,-179.9386,31.7913,-4683.1434
C00577=-91.047,9.690,24.657,179.1672,31.6940,-4686.0750
C00578=-90.755,13.981,24.767,174.6081,29.9498,-4688.7577
C00579=-91.008,16.781,25.041,167.9432,21.7872,-4690.4474
C00580=-91.772,18.686,25.406,169.1360,11.0995,-4691.5089
C00581=-92.865,20.265,25.771,173.6100,5.1205,-4692.3101
C00582=-94.037,21.871,26.043,176.8157,3.0731,-4693.0930
C00583=-94.948,23.861,26.175,178.6786,2.3162,-4694.1066
C00584=-95.323,26.720,26.245,179.7166,0.9262,-4695.6587
C00585=-95.074,30.093,26.301,-179.9821,-0.1326,-4697.5637
C00586=-94.189,33.476,26.358,-179.9972,0.0435,-4699.5659
C00587=-93.020,36.693,26.395,179.9979,0.0053,-4701.5274
C00588=-91.721,39.829,26.395,179.9977,0.0053,-4703.4725
C00589=-90.273,42.931,26.358,179.9983,0.0436,-4705.4343
C00590=-88.507,45.948,26.301,179.9790,-0.1336,-4707.4359
C00591=-86.297,48.509,26.245,-179.7191,0.9269,-4709.3411
C00592=-84.010,50.266,26.175,-178.6733,2.3167,-4710.8935
C00593=-81.959,51.029,26.043,-176.8139,3.0727,-4711.9071
C00594=-79.995,51.336,25.771,-173.6111,5.1213,-4712.6899
C00595=-78.105,51.679,25.406,-169.1359,11.0962,-4713.4910
C00596=-76.218,52.487,25.041,-167.9434,21.7869,-4714.5530
C00597=-74.059,54.287,24.767,-174.6079,29.9481,-4716.2423
C00598=-71.231,57.528,24.657,-179.1658,31.6931,-4718.9252
C00599=-68.184,61.085,24.652,179.9356,31.7887,-4721.8567
C00600=-64.734,64.734,24.655,180.0000,31.7790,-4725.0000
C00601=-61.085,68.184,24.652,-179.9356,31.7887,-4728.1433
C00602=-57.528,71.231,24.657,179.1658,31.6931,-4731.0748
C00603=-54.287,74.059,24.767,174.6079,29.9481,-4733.7577
C00604=-52.487,76.218,25.041,167.9434,21.7869,-4735.4470
C00605=-51.679,78.105,25.406,169.1359,11.0962,-4736.5090
C00606=-51.336,79.995,25.771,173.6111,5.1213,-4737.3101
C00607=-51.029,81.959,26.043,176.8139,3.0727,-4738.0929
C00608=-50.266,84.010,26.175,178.6733,2.3167,-4739.1065
C00609=-48.509,86.297,26.245,179.7191,0.9269,-4740.6589
C00610=-45.948,88.507,26.301,-179.9790,-0.1336,-4742.5641
C00611=-42.931,90.273,26.358,-179.9983,0.0436,-4744.5657
C00612=-39.829,91.721,26.395,-179.9977,0.0053,-4746.5275
C00613=-36.693,93.020,26.395,-179.9979,0.0053,-4748.4726
C00614=-33.476,94.189,26.358,179.9972,0.0435,-4750.4341
C00615=-30.093,95.074,26.301,179.9821,-0.1326,-4752.4363
C00616=-26.720,95.323,26.245,-179.7166,0.9262,-4754.3413
C00617=-23.861,94.948,26.175,-178.6786,2.3162,-4755.8934
C00618=-21.871,94.037,26.043,-176.8157,3.0731,-4756.9070
C00619=-20.265,92.865,25.771,-173.6100,5.1205,-4757.6899
C00620=-18.686,91.772,25.406,-169.1360,11.0995,-4758.4911
C00621=-16.781,91.008,25.041,-167.9432,21.7872,-4759.5526
C00622=-13.981,90.755,24.767,-174.6081,29.9498,-4761.2423
C00623=-9.690,91.047,24.657,-179.1672,31.6940,-4763.9250
C00624=-5.020,91.408,24.652,179.9386,31.7913,-4766.8566
C00625=0.000,91.548,24.655,-180.0000,31.7764,-4770.0000
C00626=0.000,90.369,26.513,-180.0000,33.0099,-4770.0000
C00627=4.912,90.233,26.509,-179.9262,33.0210,-4773.1159
C00628=9.508,89.882,26.515,178.9946,32.9112,-4776.0385
C00629=13.759,89.629,26.645,173.5375,30.8885,-4778.7274
C00630=16.509,89.983,26.968,166.4353,20.8945,-4780.3963
C00631=18.373,90.901,27.402,169.1303,9.3354,-4781.4267
C00632=19.923,92.196,27.838,174.3403,3.7616,-4782.1938
C00633=21.502,93.597,28.166,177.5283,1.9745,-4782.9380
C00634=23.458,94.728,28.327,178.9719,1.5285,-4783.9087
C00635=26.340,95.277,28.411,179.8126,0.5486,-4785.4538
C00636=29.791,95.129,28.479,-179.9530,-0.3035,-4787.3887
C00637=33.285,94.252,28.548,-179.9987,0.0308,-4789.4506
C00638=36.628,93.045,28.594,-180.0000,0.0000,-4791.4875
C00639=39.893,91.693,28.594,-180.0000,0.0000,-4793.5125
C00640=43.110,90.182,28.548,179.9980,0.0308,-4795.5494
C00641=46.201,88.332,28.479,179.9517,-0.3033,-4797.6113
C00642=48.746,85.996,28.411,-179.8105,0.5487,-4799.5463
C00643=50.396,83.570,28.327,-178.9712,1.5238,-4801.0916
C00644=50.979,81.387,28.166,-177.5285,1.9748,-4802.0621
C00645=51.105,79.281,27.838,-174.3410,3.7642,-4802.8061
C00646=51.285,77.269,27.402,-169.1264,9.3352,-4803.5730
C00647=51.954,75.301,26.968,-166.4345,20.8949,-4804.6038
C00648=53.649,73.106,26.645,-173.5375,30.8897,-4806.2732
C00649=56.833,70.280,26.515,-178.9895,32.9101,-4808.9613
C00650=60.331,67.277,26.509,179.9267,33.0184,-4811.8843
C00651=63.901,63.901,26.513,-180.0000,33.0078,-4815.0000
C00652=67.277,60.331,26.509,-179.9267,33.0184,-4818.1157
C00653=70.280,56.833,26.515,178.9895,32.9101,-4821.0387
C00654=73.106,53.649,26.645,173.5375,30.8897,-4823.7268
C00655=75.301,51.954,26.968,166.4345,20.8949,-4825.3962
C00656=77.269,51.285,27.402,169.1264,9.3352,-4826.4270
C00657=79.281,51.105,27.838,174.3410,3.7642,-4827.1939
C00658=81.387,50.979,28.166,177.5285,1.9748,-4827.9379
C00659=83.570,50.396,28.327,178.9712,1.5238,-4828.9084
C00660=85.996,48.746,28.411,179.8105,0.5487,-4830.4537
C00661=88.332,46.201,28.479,-179.9517,-0.3033,-4832.3887
C00662=90.182,43.110,28.548,-179.9980,0.0308,-4834.4506
C00663=91.693,39.893,28.594,-180.0000,0.0000,-4836.4875
C00664=93.045,36.628,28.594,-180.0000,0.0000,-4838.5125
C00665=94.252,33.285,28.548,179.9987,0.0308,-4840.5494
C00666=95.129,29.791,28.479,179.9530,-0.3035,-4842.6113
C00667=95.277,26.340,28.411,-179.8126,0.5486,-4844.5462
C00668=94.728,23.458,28.327,-178.9719,1.5285,-4846.0913
C00669=93.597,21.502,28.166,-177.5283,1.9745,-4847.0620
C00670=92.196,19.923,27.838,-174.3403,3.7616,-4847.8062
C00671=90.901,18.373,27.402,-169.1303,9.3354,-4848.5733
C00672=89.983,16.509,26.968,-166.4353,20.8945,-4849.6037
C00673=89.629,13.759,26.645,-173.5375,30.8885,-4851.2726
C00674=89.882,9.508,26.515,-178.9946,32.9112,-4853.9615
C00675=90.233,4.912,26.509,179.9262,33.0210,-4856.8841
C00676=90.369,0.000,26.513,-180.0000,33.0099,-4860.0000
C00677=90.233,-4.912,26.509,-179.9262,33.0210,-4863.1159
C00678=89.882,-9.508,26.515,178.9946,32.9112,-4866.0385
C00679=89.629,-13.759,26.645,173.5375,30.8885,-4868.7274
C00680=89.983,-16.509,26.968,166.4353,20.8945,-4870.3963
C00681=90.901,-18.373,27.402,169.1303,9.3354,-4871.4267
C00682=92.196,-19.923,27.838,174.3403,3.7616,-4872.1938
C00683=93.597,-21.502,28.166,177.5283,1.9745,-4872.9380
C00684=94.728,-23.458,28.327,178.9719,1.5285,-4873.9087
C00685=95.277,-26.340,28.411,179.8126,0.5486,-4875.4538
C00686=95.129,-29.791,28.479,-179.9530,-0.3035,-4877.3887
C00687=94.252,-33.285,28.548,-179.9987,0.0308,-4879.4506
C00688=93.045,-36.628,28.594,-180.0000,0.0000,-4881.4875
C00689=91.693,-39.893,28.594,-180.0000,0.0000,-4883.5125
C00690=90.182,-43.110,28.548,179.9980,0.0308,-4885.5494
C00691=88.332,-46.201,28.479,179.9517,-0.3033,-4887.6113
C00692=85.996,-48.746,28.411,-179.8105,0.5487,-4889.5463
C00693=83.570,-50.396,28.327,-178.9712,1.5238,-4891.0916
C00694=81.387,-50.979,28.166,-177.5285,1.9748,-4892.0621
C00695=79.281,-51.105,27.838,-174.3410,3.7642,-4892.8061
C00696=77.269,-51.285,27.402,-169.1264,9.3352,-4893.5730
C00697=75.301,-51.954,26.968,-166.4345,20.8949,-4894.6038
C00698=73.106,-53.649,26.645,-173.5375,30.8897,-4896.2732
C00699=70.280,-56.833,26.515,-178.9895,32.9101,-4898.9613
C00700=67.277,-60.331,26.509,179.9267,33.0184,-4901.8843
C00701=63.901,-63.901,26.513,180.0000,33.0078,-4905.0000
C00702=60.331,-67.277,26.509,-179.9267,33.0184,-4908.1157
C00703=56.833,-70.280,26.515,178.9895,32.9101,-4911.0387
C00704=53.649,-73.106,26.645,173.5375,30.8897,-4913.7268
C00705=51.954,-75.301,26.968,166.4345,20.8949,-4915.3962
C00706=51.285,-77.269,27.402,169.1264,9.3352,-4916.4270
C00707=51.105,-79.281,27.838,174.3410,3.7642,-4917.1939
C00708=50.979,-81.387,28.166,177.5285,1.9748,-4917.9379
C00709=50.396,-83.570,28.327,178.9712,1.5238,-4918.9084
C00710=48.746,-85.996,28.411,179.8105,0.5487,-4920.4537
C00711=46.201,-88.332,28.479,-179.9517,-0.3033,-4922.3887
C00712=43.110,-90.182,28.548,-179.9980,0.0308,-4924.4506
C00713=39.893,-91.693,28.594,-180.0000,0.0000,-4926.4875
C00714=36.628,-93.045,28.594,-180.0000,0.0000,-4928.5125
C00715=33.285,-94.252,28.548,179.9987,0.0308,-4930.5494
C00716=29.791,-95.129,28.479,179.9530,-0.3035,-4932.6113
C00717=26.340,-95.277,28.411,-179.8126,0.5486,-4934.5462
C00718=23.458,-94.728,28.327,-178.9719,1.5285,-4936.0913
C00719=21.502,-93.597,28.166,-177.5283,1.9745,-4937.0620
C00720=19.923,-92.196,27.838,-174.3403,3.7616,-4937.8062
C00721=18.373,-90.901,27.402,-169.1303,9.3354,-4938.5733
C00722=16.509,-89.983,26.968,-166.4353,20.8945,-4939.6037
C00723=13.759,-89.629,26.645,-173.5375,30.8885,-4941.2726
C00724=9.508,-89.882,26.515,-178.9946,32.9112,-4943.9615
C00725=4.912,-90.233,26.509,179.9262,33.0210,-4946.8841
C00726=0.000,-90.369,26.513,180.0000,33.0099,-4950.0000
C00727=0.000,-90.369,26.513,180.0000,33.0099,-4950.0000
C00728=-4.912,-90.233,26.509,-179.9262,33.0210,-4953.1159
C00729=-9.508,-89.882,26.515,178.9946,32.9112,-4956.0385
C00730=-13.759,-89.629,26.645,173.5375,30.8885,-4958.7274
C00731=-16.509,-89.983,26.968,166.4353,20.8945,-4960.3963
C00732=-18.373,-90.901,27.402,169.1303,9.3354,-4961.4267
C00733=-19.923,-92.196,27.838,174.3403,3.7616,-4962.1938
C00734=-21.502,-93.597,28.166,177.5283,1.9745,-4962.9380
C00735=-23.458,-94.728,28.327,178.9719,1.5285,-4963.9087
C00736=-26.340,-95.277,28.411,179.8126,0.5486,-4965.4538
C00737=-29.791,-95.129,28.479,-179.9530,-0.3035,-4967.3887
C00738=-33.285,-94.252,28.548,-179.9987,0.0308,-4969.4506
C00739=-36.628,-93.045,28.594,-180.0000,0.0000,-4971.4875
C00740=-39.893,-91.693,28.594,-180.0000,0.0000,-4973.5125
C00741=-43.110,-90.182,28.548,179.9980,0.0308,-4975.5494
C00742=-46.201,-88.332,28.479,179.9517,-0.3033,-4977.6113
C00743=-48.746,-85.996,28.411,-179.8105,0.5487,-4979.5463
C00744=-50.396,-83.570,28.327,-178.9712,1.5238,-4981.0916
C00745=-50.979,-81.387,28.166,-177.5285,1.9748,-4982.0621
C00746=-51.105,-79.281,27.838,-174.3410,3.7642,-4982.8061
C00747=-51.285,-77.269,27.402,-169.1264,9.3352,-4983.5730
C00748=-51.954,-75.301,26.968,-166.4345,20.8949,-4984.6038
C00749=-53.649,-73.106,26.645,-173.5375,30.8897,-4986.2732
C00750=-56.833,-70.280,26.515,-178.9895,32.9101,-4988.9613
C00751=-60.331,-67.277,26.509,179.9267,33.0184,-4991.8843
C00752=-63.901,-63.901,26.513,-180.0000,33.0078,-4995.0000
C00753=-67.277,-60.331,26.509,-179.9267,33.0184,-4998.1157
C00754=-70.280,-56.833,26.515,178.9895,32.9101,-5001.0387
C00755=-73.106,-53.649,26.645,173.5375,30.8897,-5003.7268
C00756=-75.301,-51.954,26.968,166.4345,20.8949,-5005.3962
C00757=-77.269,-51.285,27.402,169.1264,9.3352,-5006.4270
C00758=-79.281,-51.105,27.838,174.3410,3.7642,-5007.1939
C00759=-81.387,-50.979,28.166,177.5285,1.9748,-5007.9379
C00760=-83.570,-50.396,28.327,178.9712,1.5238,-5008.9084
C00761=-85.996,-48.746,28.411,179.8105,0.5487,-5010.4537
C00762=-88.332,-46.201,28.479,-179.9517,-0.3033,-5012.3887
C00763=-90.182,-43.110,28.548,-179.9980,0.0308,-5014.4506
C00764=-91.693,-39.893,28.594,-180.0000,0.0000,-5016.4875
C00765=-93.045,-36.628,28.594,-180.0000,0.0000,-5018.5125
C00766=-94.252,-33.285,28.548,179.9987,0.0308,-5020.5494
C00767=-95.129,-29.791,28.479,179.9530,-0.3035,-5022.6113
C00768=-95.277,-26.340,28.411,-179.8126,0.5486,-5024.5462
C00769=-94.728,-23.458,28.327,-178.9719,1.5285,-5026.0913
C00770=-93.597,-21.502,28.166,-177.5283,1.9745,-5027.0620
C00771=-92.196,-19.923,27.838,-174.3403,3.7616,-5027.8062
C00772=-90.901,-18.373,27.402,-169.1303,9.3354,-5028.5733
C00773=-89.983,-16.509,26.968,-166.4353,20.8945,-5029.6037
C00774=-89.629,-13.759,26.645,-173.5375,30.8885,-5031.2726
C00775=-89.882,-9.508,26.515,-178.9946,32.9112,-5033.9615
C00776=-90.233,-4.912,26.509,179.9262,33.0210,-5036.8841
C00777=-90.369,0.000,26.513,-180.0000,33.0099,-5040.0000
C00778=-90.233,4.912,26.509,-179.9262,33.0210,-5043.1159
C00779=-89.882,9.508,26.515,178.9946,32.9112,-5046.0385
C00780=-89.629,13.759,26.645,173.5375,30.8885,-5048.7274
C00781=-89.983,16.509,26.968,166.4353,20.8945,-5050.3963
C00782=-90.901,18.373,27.402,169.1303,9.3354,-5051.4267
C00783=-92.196,19.923,27.838,174.3403,3.7616,-5052.1938
C00784=-93.597,21.502,28.166,177.5283,1.9745,-5052.9380
C00785=-94.728,23.458,28.327,178.9719,1.5285,-5053.9087
C00786=-95.277,26.340,28.411,179.8126,0.5486,-5055.4538
C00787=-95.129,29.791,28.479,-179.9530,-0.3035,-5057.3887
C00788=-94.252,33.285,28.548,-179.9987,0.0308,-5059.4506
C00789=-93.045,36.628,28.594,-180.0000,0.0000,-5061.4875
C00790=-91.693,39.893,28.594,-180.0000,0.0000,-5063.5125
C00791=-90.182,43.110,28.548,179.9980,0.0308,-5065.5494
C00792=-88.332,46.201,28.479,179.9517,-0.3033,-5067.6113
C00793=-85.996,48.746,28.411,-179.8105,0.5487,-5069.5463
C00794=-83.570,50.396,28.327,-178.9712,1.5238,-5071.0916
C00795=-81.387,50.979,28.166,-177.5285,1.9748,-5072.0621
C00796=-79.281,51.105,27.838,-174.3410,3.7642,-5072.8061
C00797=-77.269,51.285,27.402,-169.1264,9.3352,-5073.5730
C00798=-75.301,51.954,26.968,-166.4345,20.8949,-5074.6038
C00799=-73.106,53.649,26.645,-173.5375,30.8897,-5076.2732
C00800=-70.280,56.833,26.515,-178.9895,32.9101,-5078.9613
C00801=-67.277,60.331,26.509,179.9267,33.0184,-5081.8843
C00802=-63.901,63.901,26.513,-180.0000,33.0078,-5085.0000
C00803=-60.331,67.277,26.509,-179.9267,33.0184,-5088.1157
C00804=-56.833,70.280,26.515,178.9895,32.9101,-5091.0387
C00805=-53.649,73.106,26.645,173.5375,30.8897,-5093.7268
C00806=-51.954,75.301,26.968,166.4345,20.8949,-5095.3962
C00807=-51.285,77.269,27.402,169.1264,9.3352,-5096.4270
C00808=-51.105,79.281,27.838,174.3410,3.7642,-5097.1939
C00809=-50.979,81.387,28.166,177.5285,1.9748,-5097.9379
C00810=-50.396,83.570,28.327,178.9712,1.5238,-5098.9084
C00811=-48.746,85.996,28.411,179.8105,0.5487,-5100.4537
C00812=-46.201,88.332,28.479,-179.9517,-0.3033,-5102.3887
C00813=-43.110,90.182,28.548,-179.9980,0.0308,-5104.4506
C00814=-39.893,91.693,28.594,-180.0000,0.0000,-5106.4875
C00815=-36.628,93.045,28.594,-180.0000,0.0000,-5108.5125
C00816=-33.285,94.252,28.548,179.9987,0.0308,-5110.5494
C00817=-29.791,95.129,28.479,179.9530,-0.3035,-5112.6113
C00818=-26.340,95.277,28.411,-179.8126,0.5486,-5114.5462
C00819=-23.458,94.728,28.327,-178.9719,1.5285,-5116.0913
C00820=-21.502,93.597,28.166,-177.5283,1.9745,-5117.0620
C00821=-19.923,92.196,27.838,-174.3403,3.7616,-5117.8062
C00822=-18.373,90.901,27.402,-169.1303,9.3354,-5118.5733
C00823=-16.509,89.983,26.968,-166.4353,20.8945,-5119.6037
C00824=-13.759,89.629,26.645,-173.5375,30.8885,-5121.2726
C00825=-9.508,89.882,26.515,-178.9946,32.9112,-5123.9615
C00826=-4.912,90.233,26.509,179.9262,33.0210,-5126.8841
C00827=0.000,90.369,26.513,180.0000,33.0099,-5130.0000
C00828=0.000,89.153,28.346,180.0000,34.0969,-5130.0000
C00829=4.801,89.020,28.341,-179.9168,34.1086,-5133.0871
C00830=9.321,88.681,28.348,178.8038,33.9818,-5136.0002
C00831=13.530,88.468,28.499,172.4066,31.6332,-5138.6952
C00832=16.227,88.922,28.874,165.2292,19.6025,-5140.3419
C00833=18.049,89.999,29.382,169.5475,7.5978,-5141.3400
C00834=19.567,91.502,29.895,175.3165,2.6020,-5142.0705
C00835=21.117,93.139,30.283,178.4639,1.0211,-5142.7745
C00836=23.038,94.499,30.474,179.4358,0.7176,-5143.7009
C00837=25.943,95.229,30.574,179.9458,0.1337,-5145.2391
C00838=29.476,95.186,30.656,-179.9144,-0.4893,-5147.2060
C00839=33.085,94.318,30.738,179.9997,0.0181,-5149.3299
C00840=36.560,93.071,30.793,-180.0000,0.0000,-5151.4458
C00841=39.959,91.663,30.793,-180.0000,0.0000,-5153.5540
C00842=43.298,90.088,30.738,-179.9998,0.0128,-5155.6698
C00843=46.464,88.150,30.656,179.9130,-0.4862,-5157.7938
C00844=48.993,85.682,30.574,-179.9460,0.1365,-5159.7609
C00845=50.531,83.111,30.474,-179.4372,0.7177,-5161.2994
C00846=50.927,80.791,30.283,-178.4682,1.0199,-5162.2255
C00847=50.865,78.538,29.895,-175.3211,2.6033,-5162.9290
C00848=50.876,76.401,29.382,-169.5498,7.5993,-5163.6599
C00849=51.403,74.351,28.874,-165.2308,19.5985,-5164.6583
C00850=52.989,72.123,28.499,-172.4037,31.6349,-5166.3048
C00851=56.115,69.298,28.348,-178.8001,33.9827,-5168.9993
C00852=59.552,66.342,28.341,179.9172,34.1079,-5171.9128
C00853=63.040,63.040,28.346,180.0000,34.0966,-5175.0000
C00854=66.342,59.552,28.341,-179.9172,34.1079,-5178.0872
C00855=69.298,56.115,28.348,178.8001,33.9827,-5181.0007
C00856=72.123,52.989,28.499,172.4037,31.6349,-5183.6952
C00857=74.351,51.403,28.874,165.2308,19.5985,-5185.3417
C00858=76.401,50.876,29.382,169.5498,7.5993,-5186.3401
C00859=78.538,50.865,29.895,175.3211,2.6033,-5187.0710
C00860=80.791,50.927,30.283,178.4682,1.0199,-5187.7745
C00861=83.111,50.531,30.474,179.4372,0.7177,-5188.7006
C00862=85.682,48.993,30.574,179.9460,0.1365,-5190.2391
C00863=88.150,46.464,30.656,-179.9130,-0.4862,-5192.2062
C00864=90.088,43.298,30.738,179.9998,0.0128,-5194.3302
C00865=91.663,39.959,30.793,-180.0000,0.0000,-5196.4460
C00866=93.071,36.560,30.793,-180.0000,0.0000,-5198.5542
C00867=94.318,33.085,30.738,-179.9997,0.0181,-5200.6701
C00868=95.186,29.476,30.656,179.9144,-0.4893,-5202.7940
C00869=95.229,25.943,30.574,-179.9458,0.1337,-5204.7609
C00870=94.499,23.038,30.474,-179.4358,0.7176,-5206.2991
C00871=93.139,21.117,30.283,-178.4639,1.0211,-5207.2255
C00872=91.502,19.567,29.895,-175.3165,2.6020,-5207.9295
C00873=89.999,18.049,29.382,-169.5475,7.5978,-5208.6600
C00874=88.922,16.227,28.874,-165.2292,19.6025,-5209.6581
C00875=88.468,13.530,28.499,-172.4066,31.6332,-5211.3048
C00876=88.681,9.321,28.348,-178.8038,33.9818,-5213.9998
C00877=89.020,4.801,28.341,179.9168,34.1086,-5216.9129
C00878=89.153,0.000,28.346,180.0000,34.0969,-5220.0000
C00879=89.020,-4.801,28.341,-179.9168,34.1086,-5223.0871
C00880=88.681,-9.321,28.348,178.8038,33.9818,-5226.0002
C00881=88.468,-13.530,28.499,172.4066,31.6332,-5228.6952
C00882=88.922,-16.227,28.874,165.2292,19.6025,-5230.3419
C00883=89.999,-18.049,29.382,169.5475,7.5978,-5231.3400
C00884=91.502,-19.567,29.895,175.3165,2.6020,-5232.0705
C00885=93.139,-21.117,30.283,178.4639,1.0211,-5232.7745
C00886=94.499,-23.038,30.474,179.4358,0.7176,-5233.7009
C00887=95.229,-25.943,30.574,179.9458,0.1337,-5235.2391
C00888=95.186,-29.476,30.656,-179.9144,-0.4893,-5237.2060
C00889=94.318,-33.085,30.738,179.9997,0.0181,-5239.3299
C00890=93.071,-36.560,30.793,-180.0000,0.0000,-5241.4458
C00891=91.663,-39.959,30.793,-180.0000,0.0000,-5243.5540
C00892=90.088,-43.298,30.738,-179.9998,0.0128,-5245.6698
C00893=88.150,-46.464,30.656,179.9130,-0.4862,-5247.7938
C00894=85.682,-48.993,30.574,-179.9460,0.1365,-5249.7609
C00895=83.111,-50.531,30.474,-179.4372,0.7177,-5251.2994
C00896=80.791,-50.927,30.283,-178.4682,1.0199,-5252.2255
C00897=78.538,-50.865,29.895,-175.3211,2.6033,-5252.9290
C00898=76.401,-50.876,29.382,-169.5498,7.5993,-5253.6599
C00899=74.351,-51.403,28.874,-165.2308,19.5985,-5254.6583
C00900=72.123,-52.989,28.499,-172.4037,31.6349,-5256.3048
C00901=69.298,-56.115,28.348,-178.8001,33.9827,-5258.9993
C00902=66.342,-59.552,28.341,179.9172,34.1079,-5261.9128
C00903=63.040,-63.040,28.346,-180.0000,34.0966,-5265.0000
C00904=59.552,-66.342,28.341,-179.9172,34.1079,-5268.0872
C00905=56.115,-69.298,28.348,178.8001,33.9827,-5271.0007
C00906=52.989,-72.123,28.499,172.4037,31.6349,-5273.6952
C00907=51.403,-74.351,28.874,165.2308,19.5985,-5275.3417
C00908=50.876,-76.401,29.382,169.5498,7.5993,-5276.3401
C00909=50.865,-78.538,29.895,175.3211,2.6033,-5277.0710
C00910=50.927,-80.791,30.283,178.4682,1.0199,-5277.7745
C00911=50.531,-83.111,30.474,179.4372,0.7177,-5278.7006
C00912=48.993,-85.682,30.574,179.9460,0.1365,-5280.2391
C00913=46.464,-88.150,30.656,-179.9130,-0.4862,-5282.2062
C00914=43.298,-90.088,30.738,179.9998,0.0128,-5284.3302
C00915=39.959,-91.663,30.793,-180.0000,0.0000,-5286.4460
C00916=36.560,-93.071,30.793,-180.0000,0.0000,-5288.5542
C00917=33.085,-94.318,30.738,-179.9997,0.0181,-5290.6701
C00918=29.476,-95.186,30.656,179.9144,-0.4893,-5292.7940
C00919=25.943,-95.229,30.574,-179.9458,0.1337,-5294.7609
C00920=23.038,-94.499,30.474,-179.4358,0.7176,-5296.2991
C00921=21.117,-93.139,30.283,-178.4639,1.0211,-5297.2255
C00922=19.567,-91.502,29.895,-175.3165,2.6020,-5297.9295
C00923=18.049,-89.999,29.382,-169.5475,7.5978,-5298.6600
C00924=16.227,-88.922,28.874,-165.2292,19.6025,-5299.6581
C00925=13.530,-88.468,28.499,-172.4066,31.6332,-5301.3048
C00926=9.321,-88.681,28.348,-178.8038,33.9818,-5303.9998
C00927=4.801,-89.020,28.341,179.9168,34.1086,-5306.9129
C00928=0.000,-89.153,28.346,-180.0000,34.0969,-5310.0000
C00929=0.000,-89.153,28.346,-180.0000,34.0969,-5310.0000
C00930=-4.801,-89.020,28.341,-179.9168,34.1086,-5313.0871
C00931=-9.321,-88.681,28.348,178.8038,33.9818,-5316.0002
C00932=-13.530,-88.468,28.499,172.4066,31.6332,-5318.6952
C00933=-16.227,-88.922,28.874,165.2292,19.6025,-5320.3419
C00934=-18.049,-89.999,29.382,169.5475,7.5978,-5321.3400
C00935=-19.567,-91.502,29.895,175.3165,2.6020,-5322.0705
C00936=-21.117,-93.139,30.283,178.4639,1.0211,-5322.7745
C00937=-23.038,-94.499,30.474,179.4358,0.7176,-5323.7009
C00938=-25.943,-95.229,30.574,179.9458,0.1337,-5325.2391
C00939=-29.476,-95.186,30.656,-179.9144,-0.4893,-5327.2060
C00940=-33.085,-94.318,30.738,179.9997,0.0181,-5329.3299
C00941=-36.560,-93.071,30.793,-180.0000,0.0000,-5331.4458
C00942=-39.959,-91.663,30.793,-180.0000,0.0000,-5333.5540
C00943=-43.298,-90.088,30.738,-179.9998,0.0128,-5335.6698
C00944=-46.464,-88.150,30.656,179.9130,-0.4862,-5337.7938
C00945=-48.993,-85.682,30.574,-179.9460,0.1365,-5339.7609
C00946=-50.531,-83.111,30.474,-179.4372,0.7177,-5341.2994
C00947=-50.927,-80.791,30.283,-178.4682,1.0199,-5342.2255
C00948=-50.865,-78.538,29.895,-175.3211,2.6033,-5342.9290
C00949=-50.876,-76.401,29.382,-169.5498,7.5993,-5343.6599
C00950=-51.403,-74.351,28.874,-165.2308,19.5985,-5344.6583
C00951=-52.989,-72.123,28.499,-172.4037,31.6349,-5346.3048
C00952=-56.115,-69.298,28.348,-178.8001,33.9827,-5348.9993
C00953=-59.552,-66.342,28.341,179.9172,34.1079,-5351.9128
C00954=-63.040,-63.040,28.346,-180.0000,34.0966,-5355.0000
C00955=-66.342,-59.552,28.341,-179.9172,34.1079,-5358.0872
C00956=-69.298,-56.115,28.348,178.8001,33.9827,-5361.0007
C00957=-72.123,-52.989,28.499,172.4037,31.6349,-5363.6952
C00958=-74.351,-51.403,28.874,165.2308,19.5985,-5365.3417
C00959=-76.401,-50.876,29.382,169.5498,7.5993,-5366.3401
C00960=-78.538,-50.865,29.895,175.3211,2.6033,-5367.0710
C00961=-80.791,-50.927,30.283,178.4682,1.0199,-5367.7745
C00962=-83.111,-50.531,30.474,179.4372,0.7177,-5368.7006
C00963=-85.682,-48.993,30.574,179.9460,0.1365,-5370.2391
C00964=-88.150,-46.464,30.656,-179.9130,-0.4862,-5372.2062
C00965=-90.088,-43.298,30.738,179.9998,0.0128,-5374.3302
C00966=-91.663,-39.959,30.793,-180.0000,0.0000,-5376.4460
C00967=-93.071,-36.560,30.793,-180.0000,0.0000,-5378.5542
C00968=-94.318,-33.085,30.738,-179.9997,0.0181,-5380.6701
C00969=-95.186,-29.476,30.656,179.9144,-0.4893,-5382.7940
C00970=-95.229,-25.943,30.574,-179.9458,0.1337,-5384.7609
C00971=-94.499,-23.038,30.474,-179.4358,0.7176,-5386.2991
C00972=-93.139,-21.117,30.283,-178.4639,1.0211,-5387.2255
C00973=-91.502,-19.567,29.895,-175.3165,2.6020,-5387.9295
C00974=-89.999,-18.049,29.382,-169.5475,7.5978,-5388.6600
C00975=-88.922,-16.227,28.874,-165.2292,19.6025,-5389.6581
C00976=-88.468,-13.530,28.499,-172.4066,31.6332,-5391.3048
C00977=-88.681,-9.321,28.348,-178.8038,33.9818,-5393.9998
C00978=-89.020,-4.801,28.341,179.9168,34.1086,-5396.9129
C00979=-89.153,0.000,28.346,180.0000,34.0969,-5400.0000
C00980=-89.020,4.801,28.341,-179.9168,34.1086,-5403.0871
C00981=-88.681,9.321,28.348,178.8038,33.9818,-5406.0002
C00982=-88.468,13.530,28.499,172.4066,31.6332,-5408.6952
C00983=-88.922,16.227,28.874,165.2292,19.6025,-5410.3419
C00984=-89.999,18.049,29.382,169.5475,7.5978,-5411.3400
C00985=-91.502,19.567,29.895,175.3165,2.6020,-5412.0705
C00986=-93.139,21.117,30.283,178.4639,1.0211,-5412.7745
C00987=-94.499,23.038,30.474,179.4358,0.7176,-5413.7009
C00988=-95.229,25.943,30.574,179.9458,0.1337,-5415.2391
C00989=-95.186,29.476,30.656,-179.9144,-0.4893,-5417.2060
C00990=-94.318,33.085,30.738,179.9997,0.0181,-5419.3299
C00991=-93.071,36.560,30.793,-180.0000,0.0000,-5421.4458
C00992=-91.663,39.959,30.793,-180.0000,0.0000,-5423.5540
C00993=-90.088,43.298,30.738,-179.9998,0.0128,-5425.6698
C00994=-88.150,46.464,30.656,179.9130,-0.4862,-5427.7938
C00995=-85.682,48.993,30.574,-179.9460,0.1365,-5429.7609
C00996=-83.111,50.531,30.474,-179.4372,0.7177,-5431.2994
C00997=-80.791,50.927,30.283,-178.4682,1.0199,-5432.2255
C00998=-78.538,50.865,29.895,-175.3211,2.6033,-5432.9290
C00999=-76.401,50.876,29.382,-169.5498,7.5993,-5433.6599
C01000=-74.351,51.403,28.874,-165.2308,19.5985,-5434.6583
C01001=-72.123,52.989,28.499,-172.4037,31.6349,-5436.3048
C01002=-69.298,56.115,28.348,-178.8001,33.9827,-5438.9993
C01003=-66.342,59.552,28.341,179.9172,34.1079,-5441.9128
C01004=-63.040,63.040,28.346,180.0000,34.0966,-5445.0000
C01005=-59.552,66.342,28.341,-179.9172,34.1079,-5448.0872
C01006=-56.115,69.298,28.348,178.8001,33.9827,-5451.0007
C01007=-52.989,72.123,28.499,172.4037,31.6349,-5453.6952
C01008=-51.403,74.351,28.874,165.2308,19.5985,-5455.3417
C01009=-50.876,76.401,29.382,169.5498,7.5993,-5456.3401
C01010=-50.865,78.538,29.895,175.3211,2.6033,-5457.0710
C01011=-50.927,80.791,30.283,178.4682,1.0199,-5457.7745
C01012=-50.531,83.111,30.474,179.4372,0.7177,-5458.7006
C01013=-48.993,85.682,30.574,179.9460,0.1365,-5460.2391
C01014=-46.464,88.150,30.656,-179.9130,-0.4862,-5462.2062
C01015=-43.298,90.088,30.738,179.9998,0.0128,-5464.3302
C01016=-39.959,91.663,30.793,-180.0000,0.0000,-5466.4460
C01017=-36.560,93.071,30.793,-180.0000,0.0000,-5468.5542
C01018=-33.085,94.318,30.738,-179.9997,0.0181,-5470.6701
C01019=-29.476,95.186,30.656,179.9144,-0.4893,-5472.7940
C01020=-25.943,95.229,30.574,-179.9458,0.1337,-5474.7609
C01021=-23.038,94.499,30.474,-179.4358,0.7176,-5476.2991
C01022=-21.117,93.139,30.283,-178.4639,1.0211,-5477.2255
C01023=-19.567,91.502,29.895,-175.3165,2.6020,-5477.9295
C01024=-18.049,89.999,29.382,-169.5475,7.5978,-5478.6600
C01025=-16.227,88.922,28.874,-165.2292,19.6025,-5479.6581
C01026=-13.530,88.468,28.499,-172.4066,31.6332,-5481.3048
C01027=-9.321,88.681,28.348,-178.8038,33.9818,-5483.9998
C01028=-4.801,89.020,28.341,179.9168,34.1086,-5486.9129
C01029=0.000,89.153,28.346,-180.0000,34.0969,-5490.0000
C01030=0.000,87.904,30.157,-180.0000,35.0568,-5490.0000
C01031=4.687,87.776,30.152,-179.8975,35.0693,-5493.0565
C01032=9.129,87.447,30.160,178.5994,34.9274,-5495.9598
C01033=13.294,87.274,30.332,171.2309,32.1963,-5498.6610
C01034=15.938,87.830,30.762,164.3960,17.9884,-5500.2852
C01035=17.714,89.068,31.347,170.3040,6.0027,-5501.2483
C01036=19.200,90.783,31.942,176.4290,1.6678,-5501.9417
C01037=20.718,92.664,32.394,179.5311,0.2592,-5502.6030
C01038=22.602,94.262,32.617,-179.9450,-0.0575,-5503.4837
C01039=25.531,95.180,32.735,-179.8726,-0.2980,-5505.0155
C01040=29.149,95.246,32.831,-179.8662,-0.6721,-5507.0162
C01041=32.878,94.386,32.928,-180.0000,-0.0000,-5509.2050
C01042=36.490,93.098,32.991,-180.0000,-0.0000,-5511.4028
C01043=40.028,91.633,32.991,-180.0000,-0.0000,-5513.5971
C01044=43.493,89.989,32.928,-180.0000,-0.0000,-5515.7952
C01045=46.737,87.960,32.831,179.8655,-0.6749,-5517.9837
C01046=49.249,85.356,32.735,179.8712,-0.2926,-5519.9842
C01047=50.671,82.635,32.617,179.9485,-0.0585,-5521.5162
C01048=50.874,80.174,32.394,-179.5347,0.2613,-5522.3970
C01049=50.617,77.770,31.942,-176.4306,1.6678,-5523.0583
C01050=50.455,75.506,31.347,-170.3014,6.0013,-5523.7518
C01051=50.836,73.375,30.762,-164.3944,17.9871,-5524.7152
C01052=52.312,71.113,30.332,-171.2278,32.1987,-5526.3389
C01053=55.379,68.290,30.160,-178.5955,34.9311,-5529.0399
C01054=58.753,65.381,30.152,179.9021,35.0679,-5531.9437
C01055=62.157,62.157,30.157,-179.9951,35.0560,-5535.0000
C01056=65.381,58.753,30.152,-179.9021,35.0679,-5538.0563
C01057=68.290,55.379,30.160,178.5911,34.9274,-5540.9601
C01058=71.113,52.312,30.332,171.2332,32.1958,-5543.6611
C01059=73.375,50.836,30.762,164.3944,17.9871,-5545.2848
C01060=75.506,50.455,31.347,170.3014,6.0013,-5546.2482
C01061=77.770,50.617,31.942,176.4306,1.6678,-5546.9417
C01062=80.174,50.874,32.394,179.5347,0.2613,-5547.6030
C01063=82.635,50.671,32.617,-179.9485,-0.0585,-5548.4838
C01064=85.356,49.249,32.735,-179.8712,-0.2926,-5550.0158
C01065=87.960,46.737,32.831,-179.8655,-0.6749,-5552.0163
C01066=89.989,43.493,32.928,-180.0000,-0.0000,-5554.2048
C01067=91.633,40.028,32.991,-180.0000,-0.0000,-5556.4029
C01068=93.098,36.490,32.991,-180.0000,-0.0000,-5558.5972
C01069=94.386,32.878,32.928,-180.0000,-0.0000,-5560.7950
C01070=95.246,29.149,32.831,179.8662,-0.6721,-5562.9838
C01071=95.180,25.531,32.735,179.8726,-0.2980,-5564.9845
C01072=94.262,22.602,32.617,179.9450,-0.0575,-5566.5163
C01073=92.664,20.718,32.394,-179.5311,0.2592,-5567.3970
C01074=90.783,19.200,31.942,-176.4290,1.6678,-5568.0583
C01075=89.068,17.714,31.347,-170.3040,6.0027,-5568.7517
C01076=87.830,15.938,30.762,-164.3960,17.9884,-5569.7148
C01077=87.274,13.294,30.332,-171.2309,32.1963,-5571.3390
C01078=87.447,9.129,30.160,-178.5994,34.9274,-5574.0402
C01079=87.776,4.687,30.152,179.8975,35.0693,-5576.9435
C01080=87.904,0.000,30.157,-180.0000,35.0568,-5580.0000
C01081=87.776,-4.687,30.152,-179.9045,35.0690,-5583.0565
C01082=87.447,-9.130,30.160,178.5920,34.9269,-5585.9604
C01083=87.274,-13.294,30.332,171.2309,32.1963,-5588.6610
C01084=87.830,-15.938,30.762,164.3960,17.9884,-5590.2852
C01085=89.068,-17.714,31.347,170.3040,6.0027,-5591.2483
C01086=90.783,-19.200,31.942,176.4290,1.6678,-5591.9417
C01087=92.664,-20.718,32.394,179.5311,0.2592,-5592.6030
C01088=94.262,-22.602,32.617,-179.9450,-0.0575,-5593.4837
C01089=95.180,-25.531,32.735,-179.8726,-0.2980,-5595.0155
C01090=95.246,-29.149,32.831,-179.8662,-0.6721,-5597.0162
C01091=94.386,-32.878,32.928,-180.0000,-0.0000,-5599.2050
C01092=93.098,-36.490,32.991,-180.0000,-0.0000,-5601.4028
C01093=91.633,-40.028,32.991,-180.0000,-0.0000,-5603.5971
C01094=89.989,-43.493,32.928,-180.0000,-0.0000,-5605.7952
C01095=87.960,-46.737,32.831,179.8655,-0.6749,-5607.9837
C01096=85.356,-49.249,32.735,179.8712,-0.2926,-5609.9842
C01097=82.635,-50.671,32.617,179.9485,-0.0585,-5611.5162
C01098=80.174,-50.874,32.394,-179.5347,0.2613,-5612.3970
C01099=77.770,-50.617,31.942,-176.4306,1.6678,-5613.0583
C01100=75.506,-50.455,31.347,-170.3014,6.0013,-5613.7518
C01101=73.375,-50.836,30.762,-164.3944,17.9871,-5614.7152
C01102=71.113,-52.312,30.332,-171.2278,32.1987,-5616.3389
C01103=68.290,-55.379,30.160,-178.5955,34.9311,-5619.0399
C01104=65.381,-58.753,30.152,179.9021,35.0679,-5621.9437
C01105=62.157,-62.157,30.157,-179.9951,35.0560,-5625.0000
C01106=58.753,-65.381,30.152,-179.9021,35.0679,-5628.0563
C01107=55.379,-68.290,30.160,178.5911,34.9274,-5630.9601
C01108=52.312,-71.113,30.332,171.2332,32.1958,-5633.6611
C01109=50.836,-73.375,30.762,164.3944,17.9871,-5635.2848
C01110=50.455,-75.506,31.347,170.3014,6.0013,-5636.2482
C01111=50.617,-77.770,31.942,176.4306,1.6678,-5636.9417
C01112=50.874,-80.174,32.394,179.5347,0.2613,-5637.6030
C01113=50.671,-82.635,32.617,-179.9485,-0.0585,-5638.4838
C01114=49.249,-85.356,32.735,-179.8712,-0.2926,-5640.0158
C01115=46.737,-87.960,32.831,-179.8655,-0.6749,-5642.0163
C01116=43.493,-89.989,32.928,-180.0000,-0.0000,-5644.2048
C01117=40.028,-91.633,32.991,-180.0000,-0.0000,-5646.4029
C01118=36.490,-93.098,32.991,-180.0000,-0.0000,-5648.5972
C01119=32.878,-94.386,32.928,-180.0000,-0.0000,-5650.7950
C01120=29.149,-95.246,32.831,179.8662,-0.6721,-5652.9838
C01121=25.531,-95.180,32.735,179.8726,-0.2980,-5654.9845
C01122=22.602,-94.262,32.617,179.9450,-0.0575,-5656.5163
C01123=20.718,-92.664,32.394,-179.5311,0.2592,-5657.3970
C01124=19.200,-90.783,31.942,-176.4290,1.6678,-5658.0583
C01125=17.714,-89.068,31.347,-170.3040,6.0027,-5658.7517
C01126=15.938,-87.830,30.762,-164.3960,17.9884,-5659.7148
C01127=13.294,-87.274,30.332,-171.2309,32.1963,-5661.3390
C01128=9.129,-87.447,30.160,-178.5994,34.9274,-5664.0402
C01129=4.687,-87.776,30.152,179.8975,35.0693,-5666.9435
C01130=0.000,-87.904,30.157,180.0000,35.0568,-5670.0000
C01131=0.000,-87.904,30.157,180.0000,35.0568,-5670.0000
C01132=-4.687,-87.776,30.152,-179.9045,35.0690,-5673.0565
C01133=-9.130,-87.447,30.160,178.5920,34.9269,-5675.9604
C01134=-13.294,-87.274,30.332,171.2309,32.1963,-5678.6610
C01135=-15.938,-87.830,30.762,164.3960,17.9884,-5680.2852
C01136=-17.714,-89.068,31.347,170.3040,6.0027,-5681.2483
C01137=-19.200,-90.783,31.942,176.4290,1.6678,-5681.9417
C01138=-20.718,-92.664,32.394,179.5311,0.2592,-5682.6030
C01139=-22.602,-94.262,32.617,-179.9450,-0.0575,-5683.4837
C01140=-25.531,-95.180,32.735,-179.8726,-0.2980,-5685.0155
C01141=-29.149,-95.246,32.831,-179.8662,-0.6721,-5687.0162
C01142=-32.878,-94.386,32.928,-180.0000,-0.0000,-5689.2050
C01143=-36.490,-93.098,32.991,-180.0000,-0.0000,-5691.4028
C01144=-40.028,-91.633,32.991,-180.0000,-0.0000,-5693.5971
C01145=-43.493,-89.989,32.928,-180.0000,-0.0000,-5695.7952
C01146=-46.737,-87.960,32.831,179.8655,-0.6749,-5697.9837
C01147=-49.249,-85.356,32.735,179.8712,-0.2926,-5699.9842
C01148=-50.671,-82.635,32.617,179.9485,-0.0585,-5701.5162
C01149=-50.874,-80.174,32.394,-179.5347,0.2613,-5702.3970
C01150=-50.617,-77.770,31.942,-176.4306,1.6678,-5703.0583
C01151=-50.455,-75.506,31.347,-170.3014,6.0013,-5703.7518
C01152=-50.836,-73.375,30.762,-164.3944,17.9871,-5704.7152
C01153=-52.312,-71.113,30.332,-171.2278,32.1987,-5706.3389
C01154=-55.379,-68.290,30.160,-178.5955,34.9311,-5709.0399
C01155=-58.753,-65.381,30.152,179.9021,35.0679,-5711.9437
C01156=-62.157,-62.157,30.157,-179.9951,35.0560,-5715.0000
C01157=-65.381,-58.753,30.152,-179.9021,35.0679,-5718.0563
C01158=-68.290,-55.379,30.160,178.5911,34.9274,-5720.9601
C01159=-71.113,-52.312,30.332,171.2332,32.1958,-5723.6611
C01160=-73.375,-50.836,30.762,164.3944,17.9871,-5725.2848
C01161=-75.506,-50.455,31.347,170.3014,6.0013,-5726.2482
C01162=-77.770,-50.617,31.942,176.4306,1.6678,-5726.9417
C01163=-80.174,-50.874,32.394,179.5347,0.2613,-5727.6030
C01164=-82.635,-50.671,32.617,-179.9485,-0.0585,-5728.4838
C01165=-85.356,-49.249,32.735,-179.8712,-0.2926,-5730.0158
C01166=-87.960,-46.737,32.831,-179.8655,-0.6749,-5732.0163
C01167=-89.989,-43.493,32.928,-180.0000,-0.0000,-5734.2048
C01168=-91.633,-40.028,32.991,-180.0000,-0.0000,-5736.4029
C01169=-93.098,-36.490,32.991,-180.0000,-0.0000,-5738.5972
C01170=-94.386,-32.878,32.928,-180.0000,-0.0000,-5740.7950
C01171=-95.246,-29.149,32.831,179.8662,-0.6721,-5742.9838
C01172=-95.180,-25.531,32.735,179.8726,-0.2980,-5744.9845
C01173=-94.262,-22.602,32.617,179.9450,-0.0575,-5746.5163
C01174=-92.664,-20.718,32.394,-179.5311,0.2592,-5747.3970
C01175=-90.783,-19.200,31.942,-176.4290,1.6678,-5748.0583
C01176=-89.068,-17.714,31.347,-170.3040,6.0027,-5748.7517
C01177=-87.830,-15.938,30.762,-164.3960,17.9884,-5749.7148
C01178=-87.274,-13.294,30.332,-171.2309,32.1963,-5751.3390
C01179=-87.447,-9.129,30.160,-178.5994,34.9274,-5754.0402
C01180=-87.776,-4.687,30.152,179.8975,35.0693,-5756.9435
C01181=-87.904,0.000,30.157,-180.0000,35.0568,-5760.0000
C01182=-87.776,4.687,30.152,-179.9045,35.0690,-5763.0565
C01183=-87.447,9.130,30.160,178.5920,34.9269,-5765.9604
C01184=-87.274,13.294,30.332,171.2309,32.1963,-5768.6610
C01185=-87.830,15.938,30.762,164.3960,17.9884,-5770.2852
C01186=-89.068,17.714,31.347,170.3040,6.0027,-5771.2483
C01187=-90.783,19.200,31.942,176.4290,1.6678,-5771.9417
C01188=-92.664,20.718,32.394,179.5311,0.2592,-5772.6030
C01189=-94.262,22.602,32.617,-179.9450,-0.0575,-5773.4837
C01190=-95.180,25.531,32.735,-179.8726,-0.2980,-5775.0155
C01191=-95.246,29.149,32.831,-179.8662,-0.6721,-5777.0162
C01192=-94.386,32.878,32.928,-180.0000,-0.0000,-5779.2050
C01193=-93.098,36.490,32.991,-180.0000,-0.0000,-5781.4028
C01194=-91.633,40.028,32.991,-180.0000,-0.0000,-5783.5971
C01195=-89.989,43.493,32.928,-180.0000,-0.0000,-5785.7952
C01196=-87.960,46.737,32.831,179.8655,-0.6749,-5787.9837
C01197=-85.356,49.249,32.735,179.8712,-0.2926,-5789.9842
C01198=-82.635,50.671,32.617,179.9485,-0.0585,-5791.5162
C01199=-80.174,50.874,32.394,-179.5347,0.2613,-5792.3970
C01200=-77.770,50.617,31.942,-176.4306,1.6678,-5793.0583
C01201=-75.506,50.455,31.347,-170.3014,6.0013,-5793.7518
C01202=-73.375,50.836,30.762,-164.3944,17.9871,-5794.7152
C01203=-71.113,52.312,30.332,-171.2278,32.1987,-5796.3389
C01204=-68.290,55.379,30.160,-178.5955,34.9311,-5799.0399
C01205=-65.381,58.753,30.152,179.9021,35.0679,-5801.9437
C01206=-62.157,62.157,30.157,-179.9951,35.0560,-5805.0000
C01207=-58.753,65.381,30.152,-179.9021,35.0679,-5808.0563
C01208=-55.379,68.290,30.160,178.5911,34.9274,-5810.9601
C01209=-52.312,71.113,30.332,171.2332,32.1958,-5813.6611
C01210=-50.836,73.375,30.762,164.3944,17.9871,-5815.2848
C01211=-50.455,75.506,31.347,170.3014,6.0013,-5816.2482
C01212=-50.617,77.770,31.942,176.4306,1.6678,-5816.9417
C01213=-50.874,80.174,32.394,179.5347,0.2613,-5817.6030
C01214=-50.671,82.635,32.617,-179.9485,-0.0585,-5818.4838
C01215=-49.249,85.356,32.735,-179.8712,-0.2926,-5820.0158
C01216=-46.737,87.960,32.831,-179.8655,-0.6749,-5822.0163
C01217=-43.493,89.989,32.928,-180.0000,-0.0000,-5824.2048
C01218=-40.028,91.633,32.991,-180.0000,-0.0000,-5826.4029
C01219=-36.490,93.098,32.991,-180.0000,-0.0000,-5828.5972
C01220=-32.878,94.386,32.928,-180.0000,-0.0000,-5830.7950
C01221=-29.149,95.246,32.831,179.8662,-0.6721,-5832.9838
C01222=-25.531,95.180,32.735,179.8726,-0.2980,-5834.9845
C01223=-22.602,94.262,32.617,179.9450,-0.0575,-5836.5163
C01224=-20.718,92.664,32.394,-179.5311,0.2592,-5837.3970
C01225=-19.200,90.783,31.942,-176.4290,1.6678,-5838.0583
C01226=-17.714,89.068,31.347,-170.3040,6.0027,-5838.7517
C01227=-15.938,87.830,30.762,-164.3960,17.9884,-5839.7148
C01228=-13.294,87.274,30.332,-171.2309,32.1963,-5841.3390
C01229=-9.130,87.447,30.160,-178.5920,34.9269,-5844.0396
C01230=-4.687,87.776,30.152,179.9045,35.0690,-5846.9435
C01231=0.000,87.904,30.157,180.0000,35.0568,-5850.0000
C01232=0.000,86.627,31.948,180.0000,35.8947,-5850.0000
C01233=4.570,86.503,31.943,-179.8896,35.9073,-5853.0242
C01234=8.933,86.186,31.951,178.3732,35.7506,-5855.9175
C01235=13.053,86.053,32.146,170.0298,32.5775,-5858.6252
C01236=15.641,86.712,32.633,163.9561,16.1560,-5860.2250
C01237=17.370,88.113,33.299,171.2911,4.6136,-5861.1519
C01238=18.822,90.045,33.980,177.5928,0.9554,-5861.8065
C01239=20.308,92.176,34.500,-179.3523,-0.3032,-5862.4248
C01240=22.152,94.017,34.757,-179.2110,-0.7502,-5863.2580
C01241=25.107,95.129,34.893,-179.6486,-0.7251,-5864.7847
C01242=28.812,95.307,35.004,-179.8159,-0.8662,-5866.8204
C01243=32.664,94.457,35.116,-179.9998,-0.0181,-5869.0758
C01244=36.417,93.126,35.190,-179.9979,-0.0053,-5871.3580
C01245=40.099,91.601,35.190,-179.9977,-0.0052,-5873.6417
C01246=43.694,89.888,35.116,-179.9976,-0.0180,-5875.9241
C01247=47.019,87.765,35.004,179.8142,-0.8665,-5878.1796
C01248=49.513,85.019,34.893,179.6485,-0.7285,-5880.2155
C01249=50.816,82.144,34.757,179.2111,-0.7508,-5881.7418
C01250=50.818,79.538,34.500,179.3519,-0.3053,-5882.5751
C01251=50.362,76.980,33.980,-177.5895,0.9541,-5883.1936
C01252=50.022,74.588,33.299,-171.2890,4.6171,-5883.8475
C01253=50.255,72.374,32.633,-163.9525,16.1553,-5884.7753
C01254=51.619,70.079,32.146,-170.0305,32.5797,-5886.3747
C01255=54.626,67.259,31.951,-178.3760,35.7490,-5889.0826
C01256=57.935,64.399,31.943,179.8882,35.9085,-5891.9754
C01257=61.254,61.254,31.948,180.0000,35.8962,-5895.0000
C01258=64.398,57.936,31.943,-179.8875,35.9085,-5898.0237
C01259=67.259,54.626,31.951,178.3760,35.7490,-5900.9174
C01260=70.079,51.619,32.146,170.0305,32.5797,-5903.6253
C01261=72.374,50.255,32.633,163.9525,16.1553,-5905.2247
C01262=74.588,50.022,33.299,171.2890,4.6171,-5906.1525
C01263=76.980,50.362,33.980,177.5895,0.9541,-5906.8064
C01264=79.538,50.818,34.500,-179.3519,-0.3053,-5907.4249
C01265=82.144,50.816,34.757,-179.2111,-0.7508,-5908.2582
C01266=85.019,49.513,34.893,-179.6485,-0.7285,-5909.7845
C01267=87.765,47.019,35.004,-179.8142,-0.8665,-5911.8204
C01268=89.888,43.694,35.116,179.9976,-0.0180,-5914.0759
C01269=91.601,40.099,35.190,179.9977,-0.0052,-5916.3583
C01270=93.126,36.417,35.190,179.9979,-0.0053,-5918.6420
C01271=94.457,32.664,35.116,179.9998,-0.0181,-5920.9242
C01272=95.307,28.812,35.004,179.8159,-0.8662,-5923.1796
C01273=95.129,25.107,34.893,179.6486,-0.7251,-5925.2153
C01274=94.017,22.152,34.757,179.2110,-0.7502,-5926.7420
C01275=92.176,20.308,34.500,179.3523,-0.3032,-5927.5752
C01276=90.045,18.822,33.980,-177.5928,0.9554,-5928.1935
C01277=88.113,17.370,33.299,-171.2911,4.6136,-5928.8481
C01278=86.712,15.641,32.633,-163.9561,16.1560,-5929.7750
C01279=86.053,13.053,32.146,-170.0298,32.5775,-5931.3748
C01280=86.186,8.933,31.951,-178.3732,35.7506,-5934.0825
C01281=86.503,4.570,31.943,179.8896,35.9073,-5936.9758
C01282=86.627,0.000,31.948,-180.0000,35.8947,-5940.0000
C01283=86.503,-4.570,31.943,-179.8896,35.9073,-5943.0242
C01284=86.186,-8.933,31.951,178.3732,35.7506,-5945.9175
C01285=86.053,-13.053,32.146,170.0298,32.5775,-5948.6252
C01286=86.712,-15.641,32.633,163.9561,16.1560,-5950.2250
C01287=88.113,-17.370,33.299,171.2911,4.6136,-5951.1519
C01288=90.045,-18.822,33.980,177.5928,0.9554,-5951.8065
C01289=92.176,-20.308,34.500,-179.3523,-0.3032,-5952.4248
C01290=94.017,-22.152,34.757,-179.2110,-0.7502,-5953.2580
C01291=95.129,-25.107,34.893,-179.6486,-0.7251,-5954.7847
C01292=95.307,-28.812,35.004,-179.8159,-0.8662,-5956.8204
C01293=94.457,-32.664,35.116,-179.9998,-0.0181,-5959.0758
C01294=93.126,-36.417,35.190,-179.9979,-0.0053,-5961.3580
C01295=91.601,-40.099,35.190,-179.9977,-0.0052,-5963.6417
C01296=89.888,-43.694,35.116,-179.9976,-0.0180,-5965.9241
C01297=87.765,-47.019,35.004,179.8142,-0.8665,-5968.1796
C01298=85.019,-49.513,34.893,179.6485,-0.7285,-5970.2155
C01299=82.144,-50.816,34.757,179.2111,-0.7508,-5971.7418
C01300=79.538,-50.818,34.500,179.3519,-0.3053,-5972.5751
C01301=76.980,-50.362,33.980,-177.5895,0.9541,-5973.1936
C01302=74.588,-50.022,33.299,-171.2890,4.6171,-5973.8475
C01303=72.374,-50.255,32.633,-163.9525,16.1553,-5974.7753
C01304=70.079,-51.619,32.146,-170.0305,32.5797,-5976.3747
C01305=67.259,-54.626,31.951,-178.3760,35.7490,-5979.0826
C01306=64.399,-57.935,31.943,179.8882,35.9085,-5981.9754
C01307=61.254,-61.254,31.948,-180.0000,35.8962,-5985.0000
C01308=57.936,-64.398,31.943,-179.8875,35.9085,-5988.0237
C01309=54.626,-67.259,31.951,178.3760,35.7490,-5990.9174
C01310=51.619,-70.079,32.146,170.0305,32.5797,-5993.6253
C01311=50.255,-72.374,32.633,163.9525,16.1553,-5995.2247
C01312=50.022,-74.588,33.299,171.2890,4.6171,-5996.1525
C01313=50.362,-76.980,33.980,177.5895,0.9541,-5996.8064
C01314=50.818,-79.538,34.500,-179.3519,-0.3053,-5997.4249
C01315=50.816,-82.144,34.757,-179.2111,-0.7508,-5998.2582
C01316=49.513,-85.019,34.893,-179.6485,-0.7285,-5999.7845
C01317=47.019,-87.765,35.004,-179.8142,-0.8665,-6001.8204
C01318=43.694,-89.888,35.116,179.9976,-0.0180,-6004.0759
C01319=40.099,-91.601,35.190,179.9977,-0.0052,-6006.3583
C01320=36.417,-93.126,35.190,179.9979,-0.0053,-6008.6420
C01321=32.664,-94.457,35.116,179.9998,-0.0181,-6010.9242
C01322=28.812,-95.307,35.004,179.8159,-0.8662,-6013.1796
C01323=25.107,-95.129,34.893,179.6486,-0.7251,-6015.2153
C01324=22.152,-94.017,34.757,179.2110,-0.7502,-6016.7420
C01325=20.308,-92.176,34.500,179.3523,-0.3032,-6017.5752
C01326=18.822,-90.045,33.980,-177.5928,0.9554,-6018.1935
C01327=17.370,-88.113,33.299,-171.2911,4.6136,-6018.8481
C01328=15.641,-86.712,32.633,-163.9561,16.1560,-6019.7750
C01329=13.053,-86.053,32.146,-170.0298,32.5775,-6021.3748
C01330=8.933,-86.186,31.951,-178.3732,35.7506,-6024.0825
C01331=4.570,-86.503,31.943,179.8896,35.9073,-6026.9758
C01332=0.000,-86.627,31.948,-180.0000,35.8947,-6030.0000
C01333=0.000,-86.627,31.948,-180.0000,35.8947,-6030.0000
C01334=-4.570,-86.503,31.943,-179.8896,35.9073,-6033.0242
C01335=-8.933,-86.186,31.951,178.3732,35.7506,-6035.9175
C01336=-13.053,-86.053,32.146,170.0298,32.5775,-6038.6252
C01337=-15.641,-86.712,32.633,163.9561,16.1560,-6040.2250
C01338=-17.370,-88.113,33.299,171.2911,4.6136,-6041.1519
C01339=-18.822,-90.045,33.980,177.5928,0.9554,-6041.8065
C01340=-20.308,-92.176,34.500,-179.3523,-0.3032,-6042.4248
C01341=-22.152,-94.017,34.757,-179.2110,-0.7502,-6043.2580
C01342=-25.107,-95.129,34.893,-179.6486,-0.7251,-6044.7847
C01343=-28.812,-95.307,35.004,-179.8159,-0.8662,-6046.8204
C01344=-32.664,-94.457,35.116,-179.9998,-0.0181,-6049.0758
C01345=-36.417,-93.126,35.190,-179.9979,-0.0053,-6051.3580
C01346=-40.099,-91.601,35.190,-179.9977,-0.0052,-6053.6417
C01347=-43.694,-89.888,35.116,-179.9976,-0.0180,-6055.9241
C01348=-47.019,-87.765,35.004,179.8142,-0.8665,-6058.1796
C01349=-49.513,-85.019,34.893,179.6485,-0.7285,-6060.2155
C01350=-50.816,-82.144,34.757,179.2111,-0.7508,-6061.7418
C01351=-50.818,-79.538,34.500,179.3519,-0.3053,-6062.5751
C01352=-50.362,-76.980,33.980,-177.5895,0.9541,-6063.1936
C01353=-50.022,-74.588,33.299,-171.2890,4.6171,-6063.8475
C01354=-50.255,-72.374,32.633,-163.9525,16.1553,-6064.7753
C01355=-51.619,-70.079,32.146,-170.0305,32.5797,-6066.3747
C01356=-54.626,-67.259,31.951,-178.3760,35.7490,-6069.0826
C01357=-57.935,-64.399,31.943,179.8882,35.9085,-6071.9754
C01358=-61.254,-61.254,31.948,-180.0000,35.8962,-6075.0000
C01359=-64.398,-57.936,31.943,-179.8875,35.9085,-6078.0237
C01360=-67.259,-54.626,31.951,178.3760,35.7490,-6080.9174
C01361=-70.079,-51.619,32.146,170.0305,32.5797,-6083.6253
C01362=-72.374,-50.255,32.633,163.9525,16.1553,-6085.2247
C01363=-74.588,-50.022,33.299,171.2890,4.6171,-6086.1525
C01364=-76.980,-50.362,33.980,177.5895,0.9541,-6086.8064
C01365=-79.538,-50.818,34.500,-179.3519,-0.3053,-6087.4249
C01366=-82.144,-50.816,34.757,-179.2111,-0.7508,-6088.2582
C01367=-85.019,-49.513,34.893,-179.6485,-0.7285,-6089.7845
C01368=-87.765,-47.019,35.004,-179.8142,-0.8665,-6091.8204
C01369=-89.888,-43.694,35.116,179.9976,-0.0180,-6094.0759
C01370=-91.601,-40.099,35.190,179.9977,-0.0052,-6096.3583
C01371=-93.126,-36.417,35.190,179.9979,-0.0053,-6098.6420
C01372=-94.457,-32.664,35.116,179.9998,-0.0181,-6100.9242
C01373=-95.307,-28.812,35.004,179.8159,-0.8662,-6103.1796
C01374=-95.129,-25.107,34.893,179.6486,-0.7251,-6105.2153
C01375=-94.017,-22.152,34.757,179.2110,-0.7502,-6106.7420
C01376=-92.176,-20.308,34.500,179.3523,-0.3032,-6107.5752
C01377=-90.045,-18.822,33.980,-177.5928,0.9554,-6108.1935
C01378=-88.113,-17.370,33.299,-171.2911,4.6136,-6108.8481
C01379=-86.712,-15.641,32.633,-163.9561,16.1560,-6109.7750
C01380=-86.053,-13.053,32.146,-170.0298,32.5775,-6111.3748
C01381=-86.186,-8.933,31.951,-178.3732,35.7506,-6114.0825
C01382=-86.503,-4.570,31.943,179.8896,35.9073,-6116.9758
C01383=-86.627,0.000,31.948,180.0000,35.8947,-6120.0000
C01384=-86.503,4.570,31.943,-179.8896,35.9073,-6123.0242
C01385=-86.186,8.933,31.951,178.3732,35.7506,-6125.9175
C01386=-86.053,13.053,32.146,170.0298,32.5775,-6128.6252
C01387=-86.712,15.641,32.633,163.9561,16.1560,-6130.2250
C01388=-88.113,17.370,33.299,171.2911,4.6136,-6131.1519
C01389=-90.045,18.822,33.980,177.5928,0.9554,-6131.8065
C01390=-92.176,20.308,34.500,-179.3523,-0.3032,-6132.4248
C01391=-94.017,22.152,34.757,-179.2110,-0.7502,-6133.2580
C01392=-95.129,25.107,34.893,-179.6486,-0.7251,-6134.7847
C01393=-95.307,28.812,35.004,-179.8159,-0.8662,-6136.8204
C01394=-94.457,32.664,35.116,-179.9998,-0.0181,-6139.0758
C01395=-93.126,36.417,35.190,-179.9979,-0.0053,-6141.3580
C01396=-91.601,40.099,35.190,-179.9977,-0.0052,-6143.6417
C01397=-89.888,43.694,35.116,-179.9976,-0.0180,-6145.9241
C01398=-87.765,47.019,35.004,179.8142,-0.8665,-6148.1796
C01399=-85.019,49.513,34.893,179.6485,-0.7285,-6150.2155
C01400=-82.144,50.816,34.757,179.2111,-0.7508,-6151.7418
C01401=-79.538,50.818,34.500,179.3519,-0.3053,-6152.5751
C01402=-76.980,50.362,33.980,-177.5895,0.9541,-6153.1936
C01403=-74.588,50.022,33.299,-171.2890,4.6171,-6153.8475
C01404=-72.374,50.255,32.633,-163.9525,16.1553,-6154.7753
C01405=-70.079,51.619,32.146,-170.0305,32.5797,-6156.3747
C01406=-67.259,54.626,31.951,-178.3760,35.7490,-6159.0826
C01407=-64.399,57.935,31.943,179.8882,35.9085,-6161.9754
C01408=-61.254,61.254,31.948,180.0000,35.8962,-6165.0000
C01409=-57.936,64.398,31.943,-179.8875,35.9085,-6168.0237
C01410=-54.626,67.259,31.951,178.3760,35.7490,-6170.9174
C01411=-51.619,70.079,32.146,170.0305,32.5797,-6173.6253
C01412=-50.255,72.374,32.633,163.9525,16.1553,-6175.2247
C01413=-50.022,74.588,33.299,171.2890,4.6171,-6176.1525
C01414=-50.362,76.980,33.980,177.5895,0.9541,-6176.8064
C01415=-50.818,79.538,34.500,-179.3519,-0.3053,-6177.4249
C01416=-50.816,82.144,34.757,-179.2111,-0.7508,-6178.2582
C01417=-49.513,85.019,34.893,-179.6485,-0.7285,-6179.7845
C01418=-47.019,87.765,35.004,-179.8142,-0.8665,-6181.8204
C01419=-43.694,89.888,35.116,179.9976,-0.0180,-6184.0759
C01420=-40.099,91.601,35.190,179.9977,-0.0052,-6186.3583
C01421=-36.417,93.126,35.190,179.9979,-0.0053,-6188.6420
C01422=-32.664,94.457,35.116,179.9998,-0.0181,-6190.9242
C01423=-28.812,95.307,35.004,179.8159,-0.8662,-6193.1796
C01424=-25.107,95.129,34.893,179.6486,-0.7251,-6195.2153
C01425=-22.152,94.017,34.757,179.2110,-0.7502,-6196.7420
C01426=-20.308,92.176,34.500,179.3523,-0.3032,-6197.5752
C01427=-18.822,90.045,33.980,-177.5928,0.9554,-6198.1935
C01428=-17.370,88.113,33.299,-171.2911,4.6136,-6198.8481
C01429=-15.641,86.712,32.633,-163.9561,16.1560,-6199.7750
C01430=-13.053,86.053,32.146,-170.0298,32.5775,-6201.3748
C01431=-8.933,86.186,31.951,-178.3732,35.7506,-6204.0825
C01432=-4.570,86.503,31.943,179.8896,35.9073,-6206.9758
C01433=0.000,86.627,31.948,-180.0000,35.8947,-6210.0000
C01434=0.000,85.325,33.722,-180.0000,36.6281,-6210.0000
C01435=4.451,85.206,33.716,-179.8737,36.6409,-6212.9903
C01436=8.733,84.900,33.725,178.1463,36.4598,-6215.8729
C01437=12.808,84.808,33.943,168.8261,32.7893,-6218.5881
C01438=15.338,85.570,34.490,163.9088,14.2031,-6220.1621
C01439=17.019,87.137,35.239,172.4198,3.4506,-6221.0515
C01440=18.435,89.289,36.009,178.7364,0.4238,-6221.6656
C01441=19.887,91.675,36.600,-178.2531,-0.7002,-6222.2395
C01442=21.692,93.766,36.894,-178.4010,-1.3423,-6223.0258
C01443=24.671,95.076,37.049,-179.3934,-1.1510,-6224.5467
C01444=28.465,95.370,37.176,-179.7578,-1.0519,-6226.6187
C01445=32.445,94.529,37.304,-179.9997,-0.0362,-6228.9437
C01446=36.342,93.155,37.389,-179.9979,-0.0053,-6231.3119
C01447=40.172,91.569,37.389,-179.9977,-0.0052,-6233.6874
C01448=43.901,89.784,37.304,179.9971,-0.0333,-6236.0569
C01449=47.309,87.565,37.176,179.7616,-1.0536,-6238.3812
C01450=49.784,84.674,37.049,179.3922,-1.1484,-6240.4534
C01451=50.965,81.641,36.894,178.3995,-1.3439,-6241.9748
C01452=50.762,78.886,36.600,178.2560,-0.6999,-6242.7607
C01453=50.101,76.172,36.009,-178.7370,0.4261,-6243.3343
C01454=49.580,73.649,35.239,-172.4189,3.4541,-6243.9482
C01455=49.662,71.353,34.490,-163.9057,14.2058,-6244.8381
C01456=50.912,69.025,33.943,-168.8287,32.7883,-6246.4120
C01457=53.858,66.209,33.725,-178.1431,36.4603,-6249.1268
C01458=57.102,63.397,33.716,179.8751,36.6399,-6252.0095
C01459=60.334,60.334,33.722,-180.0000,36.6307,-6255.0000
C01460=63.397,57.102,33.716,-179.8751,36.6399,-6257.9905
C01461=66.209,53.858,33.725,178.1431,36.4603,-6260.8732
C01462=69.025,50.912,33.943,168.8287,32.7883,-6263.5880
C01463=71.353,49.662,34.490,163.9057,14.2058,-6265.1619
C01464=73.649,49.580,35.239,172.4189,3.4541,-6266.0518
C01465=76.172,50.101,36.009,178.7370,0.4261,-6266.6657
C01466=78.886,50.762,36.600,-178.2560,-0.6999,-6267.2393
C01467=81.641,50.965,36.894,-178.3995,-1.3439,-6268.0252
C01468=84.674,49.784,37.049,-179.3922,-1.1484,-6269.5466
C01469=87.565,47.309,37.176,-179.7616,-1.0536,-6271.6188
C01470=89.784,43.901,37.304,-179.9971,-0.0333,-6273.9431
C01471=91.569,40.172,37.389,179.9977,-0.0052,-6276.3126
C01472=93.155,36.342,37.389,179.9979,-0.0053,-6278.6881
C01473=94.529,32.445,37.304,179.9997,-0.0362,-6281.0563
C01474=95.370,28.465,37.176,179.7578,-1.0519,-6283.3813
C01475=95.076,24.671,37.049,179.3934,-1.1510,-6285.4533
C01476=93.766,21.692,36.894,178.4010,-1.3423,-6286.9742
C01477=91.675,19.887,36.600,178.2531,-0.7002,-6287.7605
C01478=89.289,18.435,36.009,-178.7364,0.4238,-6288.3344
C01479=87.137,17.019,35.239,-172.4198,3.4506,-6288.9485
C01480=85.570,15.338,34.490,-163.9088,14.2031,-6289.8379
C01481=84.808,12.808,33.943,-168.8261,32.7893,-6291.4119
C01482=84.900,8.733,33.725,-178.1463,36.4598,-6294.1271
C01483=85.206,4.451,33.716,179.8737,36.6409,-6297.0097
C01484=85.325,0.000,33.722,-180.0000,36.6281,-6300.0000
C01485=85.206,-4.451,33.716,-179.8737,36.6409,-6302.9903
C01486=84.900,-8.733,33.725,178.1463,36.4598,-6305.8729
C01487=84.808,-12.808,33.943,168.8327,32.7900,-6308.5881
C01488=85.570,-15.338,34.490,163.9088,14.2031,-6310.1621
C01489=87.137,-17.019,35.239,172.4198,3.4506,-6311.0515
C01490=89.289,-18.435,36.009,178.7364,0.4238,-6311.6656
C01491=91.675,-19.887,36.600,-178.2531,-0.7002,-6312.2395
C01492=93.766,-21.692,36.894,-178.4010,-1.3423,-6313.0258
C01493=95.076,-24.671,37.049,-179.3934,-1.1510,-6314.5467
C01494=95.370,-28.465,37.176,-179.7578,-1.0519,-6316.6187
C01495=94.529,-32.445,37.304,-179.9997,-0.0362,-6318.9437
C01496=93.155,-36.342,37.389,-179.9979,-0.0053,-6321.3119
C01497=91.569,-40.172,37.389,-179.9977,-0.0052,-6323.6874
C01498=89.784,-43.901,37.304,179.9971,-0.0333,-6326.0569
C01499=87.565,-47.309,37.176,179.7616,-1.0536,-6328.3812
C01500=84.674,-49.784,37.049,179.3922,-1.1484,-6330.4534
C01501=81.641,-50.965,36.894,178.3995,-1.3439,-6331.9748
C01502=78.886,-50.762,36.600,178.2560,-0.6999,-6332.7607
C01503=76.172,-50.101,36.009,-178.7370,0.4261,-6333.3343
C01504=73.649,-49.580,35.239,-172.4189,3.4541,-6333.9482
C01505=71.353,-49.662,34.490,-163.9057,14.2058,-6334.8381
C01506=69.025,-50.912,33.943,-168.8287,32.7883,-6336.4120
C01507=66.209,-53.858,33.725,-178.1431,36.4603,-6339.1268
C01508=63.397,-57.102,33.716,179.8751,36.6399,-6342.0095
C01509=60.334,-60.334,33.722,180.0000,36.6307,-6345.0000
C01510=57.102,-63.397,33.716,-179.8751,36.6399,-6347.9905
C01511=53.858,-66.209,33.725,178.1431,36.4603,-6350.8732
C01512=50.912,-69.025,33.943,168.8287,32.7883,-6353.5880
C01513=49.662,-71.353,34.490,163.9057,14.2058,-6355.1619
C01514=49.580,-73.649,35.239,172.4189,3.4541,-6356.0518
C01515=50.101,-76.172,36.009,178.7370,0.4261,-6356.6657
C01516=50.762,-78.886,36.600,-178.2560,-0.6999,-6357.2393
C01517=50.965,-81.641,36.894,-178.3995,-1.3439,-6358.0252
C01518=49.784,-84.674,37.049,-179.3922,-1.1484,-6359.5466
C01519=47.309,-87.565,37.176,-179.7616,-1.0536,-6361.6188
C01520=43.901,-89.784,37.304,-179.9971,-0.0333,-6363.9431
C01521=40.172,-91.569,37.389,179.9977,-0.0052,-6366.3126
C01522=36.342,-93.155,37.389,179.9979,-0.0053,-6368.6881
C01523=32.445,-94.529,37.304,179.9997,-0.0362,-6371.0563
C01524=28.465,-95.370,37.176,179.7578,-1.0519,-6373.3813
C01525=24.671,-95.076,37.049,179.3934,-1.1510,-6375.4533
C01526=21.692,-93.766,36.894,178.4010,-1.3423,-6376.9742
C01527=19.887,-91.675,36.600,178.2531,-0.7002,-6377.7605
C01528=18.435,-89.289,36.009,-178.7364,0.4238,-6378.3344
C01529=17.019,-87.137,35.239,-172.4198,3.4506,-6378.9485
C01530=15.338,-85.570,34.490,-163.9088,14.2031,-6379.8379
C01531=12.808,-84.808,33.943,-168.8261,32.7893,-6381.4119
C01532=8.733,-84.900,33.725,-178.1463,36.4598,-6384.1271
C01533=4.451,-85.206,33.716,179.8737,36.6409,-6387.0097
C01534=0.000,-85.325,33.722,180.0000,36.6281,-6390.0000
C01535=0.000,-85.325,33.722,180.0000,36.6281,-6390.0000
C01536=-4.451,-85.206,33.716,-179.8737,36.6409,-6392.9903
C01537=-8.733,-84.900,33.725,178.1463,36.4598,-6395.8729
C01538=-12.808,-84.808,33.943,168.8327,32.7900,-6398.5881
C01539=-15.338,-85.570,34.490,163.9088,14.2031,-6400.1621
C01540=-17.019,-87.137,35.239,172.4198,3.4506,-6401.0515
C01541=-18.435,-89.289,36.009,178.7364,0.4238,-6401.6656
C01542=-19.887,-91.675,36.600,-178.2531,-0.7002,-6402.2395
C01543=-21.692,-93.766,36.894,-178.4010,-1.3423,-6403.0258
C01544=-24.671,-95.076,37.049,-179.3934,-1.1510,-6404.5467
C01545=-28.465,-95.370,37.176,-179.7578,-1.0519,-6406.6187
C01546=-32.445,-94.529,37.304,-179.9997,-0.0362,-6408.9437
C01547=-36.342,-93.155,37.389,-179.9979,-0.0053,-6411.3119
C01548=-40.172,-91.569,37.389,-179.9977,-0.0052,-6413.6874
C01549=-43.901,-89.784,37.304,179.9971,-0.0333,-6416.0569
C01550=-47.309,-87.565,37.176,179.7616,-1.0536,-6418.3812
C01551=-49.784,-84.674,37.049,179.3922,-1.1484,-6420.4534
C01552=-50.965,-81.641,36.894,178.3995,-1.3439,-6421.9748
C01553=-50.762,-78.886,36.600,178.2560,-0.6999,-6422.7607
C01554=-50.101,-76.172,36.009,-178.7370,0.4261,-6423.3343
C01555=-49.580,-73.649,35.239,-172.4189,3.4541,-6423.9482
C01556=-49.662,-71.353,34.490,-163.9057,14.2058,-6424.8381
C01557=-50.912,-69.025,33.943,-168.8287,32.7883,-6426.4120
C01558=-53.858,-66.209,33.725,-178.1431,36.4603,-6429.1268
C01559=-57.102,-63.397,33.716,179.8751,36.6399,-6432.0095
C01560=-60.334,-60.334,33.722,-180.0000,36.6307,-6435.0000
C01561=-63.397,-57.102,33.716,-179.8751,36.6399,-6437.9905
C01562=-66.209,-53.858,33.725,178.1431,36.4603,-6440.8732
C01563=-69.025,-50.912,33.943,168.8287,32.7883,-6443.5880
C01564=-71.353,-49.662,34.490,163.9057,14.2058,-6445.1619
C01565=-73.649,-49.580,35.239,172.4189,3.4541,-6446.0518
C01566=-76.172,-50.101,36.009,178.7370,0.4261,-6446.6657
C01567=-78.886,-50.762,36.600,-178.2560,-0.6999,-6447.2393
C01568=-81.641,-50.965,36.894,-178.3995,-1.3439,-6448.0252
C01569=-84.674,-49.784,37.049,-179.3922,-1.1484,-6449.5466
C01570=-87.565,-47.309,37.176,-179.7616,-1.0536,-6451.6188
C01571=-89.784,-43.901,37.304,-179.9971,-0.0333,-6453.9431
C01572=-91.569,-40.172,37.389,179.9977,-0.0052,-6456.3126
C01573=-93.155,-36.342,37.389,179.9979,-0.0053,-6458.6881
C01574=-94.529,-32.445,37.304,179.9997,-0.0362,-6461.0563
C01575=-95.370,-28.465,37.176,179.7578,-1.0519,-6463.3813
C01576=-95.076,-24.671,37.049,179.3934,-1.1510,-6465.4533
C01577=-93.766,-21.692,36.894,178.4010,-1.3423,-6466.9742
C01578=-91.675,-19.887,36.600,178.2531,-0.7002,-6467.7605
C01579=-89.289,-18.435,36.009,-178.7364,0.4238,-6468.3344
C01580=-87.137,-17.019,35.239,-172.4198,3.4506,-6468.9485
C01581=-85.570,-15.338,34.490,-163.9088,14.2031,-6469.8379
C01582=-84.808,-12.808,33.943,-168.8261,32.7893,-6471.4119
C01583=-84.900,-8.733,33.725,-178.1463,36.4598,-6474.1271
C01584=-85.206,-4.451,33.716,179.8737,36.6409,-6477.0097
C01585=-85.325,0.000,33.722,-180.0000,36.6281,-6480.0000
C01586=-85.206,4.451,33.716,-179.8737,36.6409,-6482.9903
C01587=-84.900,8.733,33.725,178.1463,36.4598,-6485.8729
C01588=-84.808,12.808,33.943,168.8327,32.7900,-6488.5881
C01589=-85.570,15.338,34.490,163.9088,14.2031,-6490.1621
C01590=-87.137,17.019,35.239,172.4198,3.4506,-6491.0515
C01591=-89.289,18.435,36.009,178.7364,0.4238,-6491.6656
C01592=-91.675,19.887,36.600,-178.2531,-0.7002,-6492.2395
C01593=-93.766,21.692,36.894,-178.4010,-1.3423,-6493.0258
C01594=-95.076,24.671,37.049,-179.3934,-1.1510,-6494.5467
C01595=-95.370,28.465,37.176,-179.7578,-1.0519,-6496.6187
C01596=-94.529,32.445,37.304,-179.9997,-0.0362,-6498.9437
C01597=-93.155,36.342,37.389,-179.9979,-0.0053,-6501.3119
C01598=-91.569,40.172,37.389,-179.9977,-0.0052,-6503.6874
C01599=-89.784,43.901,37.304,179.9971,-0.0333,-6506.0569
C01600=-87.565,47.309,37.176,179.7616,-1.0536,-6508.3812
C01601=-84.674,49.784,37.049,179.3922,-1.1484,-6510.4534
C01602=-81.641,50.965,36.894,178.3995,-1.3439,-6511.9748
C01603=-78.886,50.762,36.600,178.2560,-0.6999,-6512.7607
C01604=-76.172,50.101,36.009,-178.7370,0.4261,-6513.3343
C01605=-73.649,49.580,35.239,-172.4189,3.4541,-6513.9482
C01606=-71.353,49.662,34.490,-163.9057,14.2058,-6514.8381
C01607=-69.025,50.912,33.943,-168.8287,32.7883,-6516.4120
C01608=-66.209,53.858,33.725,-178.1431,36.4603,-6519.1268
C01609=-63.397,57.102,33.716,179.8751,36.6399,-6522.0095
C01610=-60.334,60.334,33.722,-180.0000,36.6307,-6525.0000
C01611=-57.102,63.397,33.716,-179.8751,36.6399,-6527.9905
C01612=-53.858,66.209,33.725,178.1431,36.4603,-6530.8732
C01613=-50.912,69.025,33.943,168.8287,32.7883,-6533.5880
C01614=-49.662,71.353,34.490,163.9057,14.2058,-6535.1619
C01615=-49.580,73.649,35.239,172.4189,3.4541,-6536.0518
C01616=-50.101,76.172,36.009,178.7370,0.4261,-6536.6657
C01617=-50.762,78.886,36.600,-178.2560,-0.6999,-6537.2393
C01618=-50.965,81.641,36.894,-178.3995,-1.3439,-6538.0252
C01619=-49.784,84.674,37.049,-179.3922,-1.1484,-6539.5466
C01620=-47.309,87.565,37.176,-179.7616,-1.0536,-6541.6188
C01621=-43.901,89.784,37.304,-179.9971,-0.0333,-6543.9431
C01622=-40.172,91.569,37.389,179.9977,-0.0052,-6546.3126
C01623=-36.342,93.155,37.389,179.9979,-0.0053,-6548.6881
C01624=-32.445,94.529,37.304,179.9997,-0.0362,-6551.0563
C01625=-28.465,95.370,37.176,179.7578,-1.0519,-6553.3813
C01626=-24.671,95.076,37.049,179.3934,-1.1510,-6555.4533
C01627=-21.692,93.766,36.894,178.4010,-1.3423,-6556.9742
C01628=-19.887,91.675,36.600,178.2531,-0.7002,-6557.7605
C01629=-18.435,89.289,36.009,-178.7364,0.4238,-6558.3344
C01630=-17.019,87.137,35.239,-172.4198,3.4506,-6558.9485
C01631=-15.338,85.570,34.490,-163.9088,14.2031,-6559.8379
C01632=-12.808,84.808,33.943,-168.8327,32.7900,-6561.4119
C01633=-8.733,84.900,33.725,-178.1463,36.4598,-6564.1271
C01634=-4.451,85.206,33.716,179.8737,36.6409,-6567.0097
C01635=0.000,85.325,33.722,180.0000,36.6281,-6570.0000
C01636=0.000,84.003,35.480,180.0000,37.2584,-6570.0000
C01637=4.330,83.888,35.473,-179.8571,37.2713,-6572.9548
C01638=8.530,83.594,35.484,177.9021,37.0692,-6575.8263
C01639=12.558,83.543,35.726,167.6478,32.8316,-6578.5486
C01640=15.030,84.409,36.333,164.2172,12.2420,-6580.0964
C01641=16.662,86.143,37.169,173.6165,2.5084,-6580.9471
C01642=18.041,88.518,38.031,179.8324,0.0477,-6581.5198
C01643=19.458,91.164,38.697,-177.2185,-0.9486,-6582.0484
C01644=21.221,93.510,39.027,-177.5538,-1.8150,-6582.7860
C01645=24.227,95.023,39.203,-179.1127,-1.5540,-6584.3034
C01646=28.112,95.435,39.346,-179.6955,-1.2364,-6586.4132
C01647=32.220,94.603,39.491,179.9985,-0.0489,-6588.8079
C01648=36.266,93.184,39.587,-179.9979,-0.0053,-6591.2653
C01649=40.247,91.535,39.587,179.9971,-0.0076,-6593.7346
C01650=44.111,89.678,39.491,179.9997,-0.0512,-6596.1917
C01651=47.604,87.360,39.346,179.6949,-1.2364,-6598.5867
C01652=50.060,84.322,39.203,179.1149,-1.5518,-6600.6966
C01653=51.116,81.128,39.027,177.5559,-1.8116,-6602.2136
C01654=50.704,78.221,38.697,177.2195,-0.9491,-6602.9519
C01655=49.835,75.348,38.031,-179.8330,0.0487,-6603.4806
C01656=49.130,72.694,37.169,-173.6149,2.5069,-6604.0527
C01657=49.058,70.314,36.333,-164.2153,12.2381,-6604.9034
C01658=50.194,67.954,35.726,-167.6473,32.8330,-6606.4513
C01659=53.078,65.141,35.484,-177.8974,37.0682,-6609.1737
C01660=56.256,62.380,35.473,179.8597,37.2688,-6612.0450
C01661=59.399,59.399,35.480,180.0000,37.2595,-6615.0000
C01662=62.380,56.256,35.473,-179.8597,37.2688,-6617.9550
C01663=65.141,53.078,35.484,177.8974,37.0682,-6620.8263
C01664=67.954,50.194,35.726,167.6473,32.8330,-6623.5487
C01665=70.314,49.058,36.333,164.2153,12.2381,-6625.0966
C01666=72.694,49.130,37.169,173.6149,2.5069,-6625.9473
C01667=75.348,49.835,38.031,179.8330,0.0487,-6626.5194
C01668=78.221,50.704,38.697,-177.2195,-0.9491,-6627.0481
C01669=81.128,51.116,39.027,-177.5559,-1.8116,-6627.7864
C01670=84.322,50.060,39.203,-179.1149,-1.5518,-6629.3034
C01671=87.360,47.604,39.346,-179.6949,-1.2364,-6631.4133
C01672=89.678,44.111,39.491,-179.9997,-0.0512,-6633.8083
C01673=91.535,40.247,39.587,-179.9971,-0.0076,-6636.2654
C01674=93.184,36.266,39.587,179.9979,-0.0053,-6638.7347
C01675=94.603,32.220,39.491,-179.9985,-0.0489,-6641.1921
C01676=95.435,28.112,39.346,179.6955,-1.2364,-6643.5868
C01677=95.023,24.227,39.203,179.1127,-1.5540,-6645.6966
C01678=93.510,21.221,39.027,177.5538,-1.8150,-6647.2140
C01679=91.164,19.458,38.697,177.2185,-0.9486,-6647.9516
C01680=88.518,18.041,38.031,-179.8324,0.0477,-6648.4802
C01681=86.143,16.662,37.169,-173.6165,2.5084,-6649.0529
C01682=84.409,15.030,36.333,-164.2172,12.2420,-6649.9036
C01683=83.543,12.558,35.726,-167.6478,32.8316,-6651.4514
C01684=83.594,8.530,35.484,-177.9021,37.0692,-6654.1737
C01685=83.888,4.330,35.473,179.8571,37.2713,-6657.0452
C01686=84.003,0.000,35.480,-180.0000,37.2584,-6660.0000
C01687=83.888,-4.330,35.473,-179.8571,37.2713,-6662.9548
C01688=83.594,-8.530,35.484,177.8949,37.0687,-6665.8263
C01689=83.543,-12.558,35.726,167.6478,32.8316,-6668.5486
C01690=84.409,-15.030,36.333,164.2172,12.2420,-6670.0964
C01691=86.143,-16.662,37.169,173.6165,2.5084,-6670.9471
C01692=88.518,-18.041,38.031,179.8324,0.0477,-6671.5198
C01693=91.164,-19.458,38.697,-177.2185,-0.9486,-6672.0484
C01694=93.510,-21.221,39.027,-177.5538,-1.8150,-6672.7860
C01695=95.023,-24.227,39.203,-179.1127,-1.5540,-6674.3034
C01696=95.435,-28.112,39.346,-179.6955,-1.2364,-6676.4132
C01697=94.603,-32.220,39.491,179.9985,-0.0489,-6678.8079
C01698=93.184,-36.266,39.587,-179.9979,-0.0053,-6681.2653
C01699=91.535,-40.247,39.587,179.9971,-0.0076,-6683.7346
C01700=89.678,-44.111,39.491,179.9997,-0.0512,-6686.1917
C01701=87.360,-47.604,39.346,179.6949,-1.2364,-6688.5867
C01702=84.322,-50.060,39.203,179.1149,-1.5518,-6690.6966
C01703=81.128,-51.116,39.027,177.5559,-1.8116,-6692.2136
C01704=78.221,-50.704,38.697,177.2195,-0.9491,-6692.9519
C01705=75.348,-49.835,38.031,-179.8330,0.0487,-6693.4806
C01706=72.694,-49.130,37.169,-173.6149,2.5069,-6694.0527
C01707=70.314,-49.058,36.333,-164.2153,12.2381,-6694.9034
C01708=67.954,-50.194,35.726,-167.6473,32.8330,-6696.4513
C01709=65.141,-53.078,35.484,-177.8974,37.0682,-6699.1737
C01710=62.380,-56.256,35.473,179.8597,37.2688,-6702.0450
C01711=59.399,-59.399,35.480,-180.0000,37.2595,-6705.0000
C01712=56.256,-62.380,35.473,-179.8597,37.2688,-6707.9550
C01713=53.078,-65.141,35.484,177.8974,37.0682,-6710.8263
C01714=50.194,-67.954,35.726,167.6473,32.8330,-6713.5487
C01715=49.058,-70.314,36.333,164.2153,12.2381,-6715.0966
C01716=49.130,-72.694,37.169,173.6149,2.5069,-6715.9473
C01717=49.835,-75.348,38.031,179.8330,0.0487,-6716.5194
C01718=50.704,-78.221,38.697,-177.2195,-0.9491,-6717.0481
C01719=51.116,-81.128,39.027,-177.5559,-1.8116,-6717.7864
C01720=50.060,-84.322,39.203,-179.1149,-1.5518,-6719.3034
C01721=47.604,-87.360,39.346,-179.6949,-1.2364,-6721.4133
C01722=44.111,-89.678,39.491,-179.9997,-0.0512,-6723.8083
C01723=40.247,-91.535,39.587,-179.9971,-0.0076,-6726.2654
C01724=36.266,-93.184,39.587,179.9979,-0.0053,-6728.7347
C01725=32.220,-94.603,39.491,-179.9985,-0.0489,-6731.1921
C01726=28.112,-95.435,39.346,179.6955,-1.2364,-6733.5868
C01727=24.227,-95.023,39.203,179.1127,-1.5540,-6735.6966
C01728=21.221,-93.510,39.027,177.5538,-1.8150,-6737.2140
C01729=19.458,-91.164,38.697,177.2185,-0.9486,-6737.9516
C01730=18.041,-88.518,38.031,-179.8324,0.0477,-6738.4802
C01731=16.662,-86.143,37.169,-173.6165,2.5084,-6739.0529
C01732=15.030,-84.409,36.333,-164.2172,12.2420,-6739.9036
C01733=12.558,-83.543,35.726,-167.6478,32.8316,-6741.4514
C01734=8.530,-83.594,35.484,-177.9021,37.0692,-6744.1737
C01735=4.330,-83.888,35.473,179.8571,37.2713,-6747.0452
C01736=0.000,-84.003,35.480,-180.0000,37.2584,-6750.0000
C01737=0.000,-84.003,35.480,-180.0000,37.2584,-6750.0000
C01738=-4.330,-83.888,35.473,-179.8571,37.2713,-6752.9548
C01739=-8.530,-83.594,35.484,177.8949,37.0687,-6755.8263
C01740=-12.558,-83.543,35.726,167.6478,32.8316,-6758.5486
C01741=-15.030,-84.409,36.333,164.2172,12.2420,-6760.0964
C01742=-16.662,-86.143,37.169,173.6165,2.5084,-6760.9471
C01743=-18.041,-88.518,38.031,179.8324,0.0477,-6761.5198
C01744=-19.458,-91.164,38.697,-177.2185,-0.9486,-6762.0484
C01745=-21.221,-93.510,39.027,-177.5538,-1.8150,-6762.7860
C01746=-24.227,-95.023,39.203,-179.1127,-1.5540,-6764.3034
